C01835=1217.029,90.676,-47.866,-178.653,5.650,148.592
C01836=1217.025,90.925,-47.885,-178.651,5.651,148.591
C01837=1217.020,91.174,-47.903,-178.648,5.652,148.591
C01838=1217.015,91.423,-47.921,-178.645,5.653,148.590
C01839=1217.010,91.673,-47.939,-178.643,5.654,148.590
C01840=1217.005,91.922,-47.957,-178.641,5.654,148.589
C01841=1217.000,92.172,-47.976,-178.638,5.655,148.588
C01842=1216.996,92.421,-47.994,-178.635,5.657,148.588
C01843=1216.991,92.670,-48.012,-178.633,5.657,148.587
C01844=1216.986,92.919,-48.030,-178.630,5.658,148.587
C01845=1216.982,93.169,-48.049,-178.628,5.659,148.586
C01846=1216.976,93.418,-48.067,-178.625,5.660,148.586
C01847=1216.971,93.667,-48.086,-178.622,5.661,148.585
C01848=1216.967,93.916,-48.104,-178.620,5.662,148.585
C01849=1216.962,94.166,-48.122,-178.617,5.662,148.584
C01850=1216.957,94.415,-48.140,-178.615,5.663,148.584
C01851=1216.952,94.664,-48.159,-178.612,5.665,148.583
C01852=1216.948,94.914,-48.178,-178.609,5.665,148.582
C01853=1216.943,95.163,-48.196,-178.607,5.666,148.582
C01854=1216.938,95.412,-48.214,-178.605,5.667,148.581
C01855=1216.932,95.661,-48.233,-178.601,5.668,148.581
C01856=1216.928,95.911,-48.251,-178.599,5.669,148.580
C01857=1216.923,96.160,-48.269,-178.597,5.670,148.579
C01858=1216.919,96.409,-48.288,-178.594,5.670,148.579
C01859=1216.914,96.659,-48.307,-178.592,5.671,148.578
C01860=1216.909,96.908,-48.325,-178.589,5.673,148.578
C01861=1216.904,97.156,-48.344,-178.587,5.674,148.577
C01862=1216.898,97.406,-48.362,-178.584,5.674,148.577
C01863=1216.894,97.656,-48.381,-178.581,5.675,148.576
C01864=1216.889,97.904,-48.399,-178.579,5.677,148.576
C01865=1216.884,98.154,-48.418,-178.576,5.677,148.575
C01866=1216.880,98.403,-48.437,-178.573,5.678,148.574
C01867=1216.875,98.652,-48.455,-178.571,5.679,148.574
C01868=1216.869,98.902,-48.473,-178.568,5.680,148.573
C01869=1216.865,99.151,-48.492,-178.566,5.681,148.573
C01870=1216.860,99.400,-48.510,-178.563,5.682,148.572
C01871=1216.856,99.650,-48.530,-178.561,5.682,148.572
C01872=1216.851,99.899,-48.548,-178.558,5.684,148.571
C01873=1216.846,100.148,-48.567,-178.555,5.685,148.571
C01874=1216.841,100.398,-48.586,-178.553,5.686,148.570
C01875=1216.836,100.646,-48.604,-178.551,5.686,148.569
C01876=1216.831,100.896,-48.623,-178.548,5.688,148.569
C01877=1216.827,101.145,-48.642,-178.545,5.689,148.568
C01878=1216.822,101.394,-48.660,-178.543,5.689,148.568
C01879=1216.817,101.643,-48.679,-178.540,5.690,148.567
C01880=1216.812,101.893,-48.698,-178.537,5.692,148.567
C01881=1216.807,102.142,-48.717,-178.535,5.692,148.566
C01882=1216.803,102.392,-48.735,-178.533,5.693,148.566
C01883=1216.797,102.641,-48.755,-178.530,5.695,148.565
C01884=1216.792,102.890,-48.773,-178.527,5.695,148.564
C01885=1216.788,103.139,-48.792,-178.525,5.696,148.564
C01886=1216.783,103.388,-48.811,-178.522,5.697,148.563
C01887=1216.779,103.638,-48.829,-178.519,5.699,148.563
C01888=1216.773,103.887,-48.849,-178.517,5.699,148.562
C01889=1216.769,104.137,-48.867,-178.514,5.700,148.562
C01890=1216.764,104.385,-48.886,-178.512,5.702,148.561
C01891=1216.759,104.634,-48.905,-178.509,5.702,148.561
C01892=1216.754,104.884,-48.924,-178.507,5.703,148.560
C01893=1216.749,105.133,-48.943,-178.504,5.704,148.559
C01894=1216.745,105.382,-48.962,-178.502,5.705,148.559
C01895=1216.740,105.631,-48.980,-178.499,5.706,148.558
C01896=1216.735,105.881,-49.000,-178.496,5.707,148.558
C01897=1216.730,106.130,-49.019,-178.494,5.708,148.557
C01898=1216.725,106.380,-49.037,-178.491,5.709,148.557
C01899=1216.721,106.628,-49.056,-178.489,5.710,148.556
C01900=1216.715,106.877,-49.075,-178.486,5.711,148.556
C01901=1216.710,107.146,-49.096,-178.483,5.712,148.555
C01902=1216.705,107.414,-49.116,-178.481,5.713,148.555
C01903=1216.700,107.683,-49.137,-178.478,5.714,148.554
C01904=1216.695,107.951,-49.157,-178.475,5.715,148.553
C01905=1216.690,108.201,-49.177,-178.472,5.716,148.553
C01906=1216.685,108.449,-49.195,-178.470,5.717,148.552
C01907=1216.681,108.699,-49.215,-178.467,5.718,148.552
C01908=1216.676,108.948,-49.233,-178.465,5.720,148.551
C01909=1216.671,109.198,-49.253,-178.462,5.720,148.551
C01910=1216.666,109.447,-49.272,-178.460,5.721,148.550
C01911=1216.662,109.696,-49.291,-178.457,5.722,148.550
C01912=1216.656,109.945,-49.310,-178.454,5.723,148.549
C01913=1216.651,110.194,-49.330,-178.452,5.724,148.549
C01914=1216.647,110.443,-49.348,-178.449,5.725,148.548
C01915=1216.642,110.693,-49.368,-178.447,5.727,148.548
C01916=1216.638,110.942,-49.387,-178.444,5.727,148.547
C01917=1216.632,111.191,-49.406,-178.442,5.728,148.546
C01918=1216.628,111.441,-49.426,-178.439,5.730,148.546
C01919=1216.623,111.689,-49.444,-178.437,5.731,148.545
C01920=1216.618,111.939,-49.464,-178.434,5.731,148.545
C01921=1216.613,112.188,-49.483,-178.431,5.733,148.544
C01922=1216.609,112.438,-49.502,-178.429,5.734,148.544
C01923=1216.603,112.686,-49.521,-178.426,5.734,148.543
C01924=1216.599,112.936,-49.541,-178.423,5.736,148.543
C01925=1216.594,113.186,-49.560,-178.421,5.737,148.542
C01926=1216.589,113.434,-49.579,-178.419,5.738,148.542
C01927=1216.585,113.684,-49.599,-178.415,5.739,148.541
C01928=1216.579,113.933,-49.618,-178.413,5.740,148.541
C01929=1216.574,114.182,-49.638,-178.411,5.741,148.540
C01930=1216.570,114.431,-49.656,-178.407,5.742,148.539
C01931=1216.565,114.680,-49.676,-178.405,5.743,148.539
C01932=1216.560,114.930,-49.696,-178.403,5.744,148.538
C01933=1216.555,115.179,-49.715,-178.400,5.745,148.538
C01934=1216.551,115.428,-49.734,-178.397,5.746,148.537
C01935=1216.546,115.677,-49.753,-178.395,5.747,148.537
C01936=1216.541,115.926,-49.773,-178.392,5.748,148.536
C01937=1216.536,116.176,-49.792,-178.390,5.749,148.536
C01938=1216.532,116.425,-49.811,-178.387,5.750,148.535
C01939=1216.527,116.673,-49.832,-178.385,5.752,148.535
C01940=1216.522,116.923,-49.851,-178.382,5.752,148.534
C01941=1216.517,117.172,-49.871,-178.379,5.754,148.534
C01942=1216.512,117.421,-49.890,-178.377,5.755,148.533
C01943=1216.507,117.670,-49.909,-178.375,5.756,148.533
C01944=1216.503,117.920,-49.929,-178.372,5.757,148.532
C01945=1216.498,118.169,-49.948,-178.369,5.758,148.532
C01946=1216.493,118.418,-49.967,-178.367,5.759,148.531
C01947=1216.488,118.667,-49.988,-178.364,5.760,148.531
C01948=1216.484,118.917,-50.007,-178.362,5.761,148.530
C01949=1216.478,119.165,-50.027,-178.359,5.762,148.529
C01950=1216.474,119.415,-50.046,-178.356,5.763,148.529
C01951=1216.470,119.664,-50.065,-178.354,5.764,148.528
C01952=1216.464,119.913,-50.085,-178.351,5.766,148.528
C01953=1216.460,120.162,-50.105,-178.348,5.766,148.527
C01954=1216.455,120.412,-50.125,-178.346,5.767,148.527
C01955=1216.450,120.661,-50.144,-178.343,5.769,148.526
C01956=1216.445,120.910,-50.164,-178.341,5.770,148.526
C01957=1216.441,121.159,-50.184,-178.338,5.770,148.525
C01958=1216.436,121.409,-50.204,-178.336,5.772,148.525
C01959=1216.430,121.657,-50.223,-178.333,5.773,148.524
C01960=1216.426,121.907,-50.243,-178.330,5.775,148.524
C01961=1216.422,122.156,-50.263,-178.328,5.775,148.523
C01962=1216.417,122.405,-50.282,-178.326,5.776,148.523
C01963=1216.412,122.654,-50.301,-178.322,5.778,148.522
C01964=1216.408,122.903,-50.322,-178.320,5.779,148.522
C01965=1216.403,123.153,-50.341,-178.318,5.779,148.521
C01966=1216.397,123.401,-50.361,-178.315,5.781,148.521
C01967=1216.393,123.650,-50.381,-178.312,5.782,148.520
C01968=1216.388,123.900,-50.401,-178.310,5.783,148.520
C01969=1216.383,124.150,-50.420,-178.307,5.784,148.519
C01970=1216.378,124.398,-50.440,-178.305,5.785,148.519
C01971=1216.374,124.647,-50.460,-178.302,5.786,148.518
C01972=1216.369,124.896,-50.480,-178.300,5.787,148.518
C01973=1216.365,125.146,-50.500,-178.297,5.789,148.517
C01974=1216.360,125.395,-50.520,-178.294,5.790,148.517
C01975=1216.355,125.644,-50.540,-178.292,5.791,148.516
C01976=1216.350,125.893,-50.559,-178.289,5.792,148.516
C01977=1216.346,126.142,-50.580,-178.287,5.793,148.515
C01978=1216.341,126.392,-50.599,-178.284,5.795,148.514
C01979=1216.336,126.641,-50.620,-178.282,5.796,148.514
C01980=1216.330,126.890,-50.640,-178.279,5.797,148.513
C01981=1216.326,127.139,-50.660,-178.276,5.798,148.513
C01982=1216.321,127.388,-50.680,-178.274,5.799,148.512
C01983=1216.317,127.637,-50.700,-178.271,5.800,148.512
C01984=1216.312,127.887,-50.720,-178.269,5.801,148.511
C01985=1216.307,128.135,-50.740,-178.266,5.803,148.511
C01986=1216.302,128.385,-50.759,-178.263,5.803,148.510
C01987=1216.298,128.634,-50.780,-178.261,5.804,148.510
C01988=1216.293,128.883,-50.800,-178.258,5.806,148.509
C01989=1216.289,129.132,-50.820,-178.256,5.807,148.509
C01990=1216.283,129.382,-50.840,-178.253,5.809,148.509
C01991=1216.278,129.630,-50.860,-178.251,5.809,148.508
C01992=1216.274,129.879,-50.881,-178.248,5.811,148.508
C01993=1216.269,130.129,-50.900,-178.245,5.812,148.507
C01994=1216.264,130.378,-50.921,-178.243,5.813,148.507
C01995=1216.260,130.627,-50.940,-178.240,5.814,148.506
C01996=1216.255,130.876,-50.961,-178.238,5.815,148.505
C01997=1216.250,131.126,-50.982,-178.235,5.816,148.505
C01998=1216.245,131.374,-51.001,-178.233,5.817,148.504
C01999=1216.240,131.623,-51.021,-178.229,5.819,148.504
C02000=1216.236,131.872,-51.042,-178.227,5.820,148.503
C02001=1216.231,132.122,-51.061,-178.225,5.822,148.503
C02002=1216.226,132.371,-51.082,-178.222,5.822,148.502
C02003=1216.221,132.620,-51.103,-178.220,5.823,148.502
C02004=1216.217,132.870,-51.122,-178.217,5.825,148.501
C02005=1216.211,133.138,-51.145,-178.214,5.826,148.501
C02006=1216.206,133.407,-51.166,-178.211,5.827,148.500
C02007=1216.201,133.675,-51.188,-178.208,5.829,148.500
C02008=1216.195,133.944,-51.210,-178.206,5.829,148.499
C02009=1216.191,134.193,-51.230,-178.203,5.831,148.499
C02010=1216.187,134.442,-51.251,-178.201,5.832,148.498
C02011=1216.182,134.691,-51.271,-178.198,5.833,148.498
C02012=1216.177,134.941,-51.291,-178.196,5.834,148.497
C02013=1216.172,135.190,-51.312,-178.193,5.836,148.497
C02014=1216.168,135.439,-51.332,-178.190,5.837,148.496
C02015=1216.163,135.688,-51.353,-178.188,5.839,148.496
C02016=1216.158,135.937,-51.373,-178.185,5.839,148.495
C02017=1216.153,136.186,-51.393,-178.182,5.841,148.495
C02018=1216.148,136.436,-51.414,-178.180,5.842,148.495
C02019=1216.144,136.685,-51.434,-178.177,5.843,148.494
C02020=1216.139,136.934,-51.455,-178.175,5.844,148.494
C02021=1216.134,137.183,-51.476,-178.172,5.846,148.493
C02022=1216.130,137.432,-51.496,-178.170,5.847,148.493
C02023=1216.125,137.681,-51.516,-178.167,5.847,148.492
C02024=1216.120,137.931,-51.537,-178.164,5.849,148.492
C02025=1216.115,138.180,-51.557,-178.162,5.850,148.491
C02026=1216.111,138.428,-51.577,-178.159,5.852,148.490
C02027=1216.106,138.678,-51.598,-178.157,5.853,148.490
C02028=1216.101,138.927,-51.619,-178.154,5.854,148.489
C02029=1216.097,139.176,-51.639,-178.152,5.855,148.489
C02030=1216.092,139.425,-51.660,-178.149,5.857,148.489
C02031=1216.087,139.674,-51.680,-178.146,5.857,148.488
C02032=1216.082,139.923,-51.701,-178.144,5.859,148.488
C02033=1216.078,140.172,-51.722,-178.141,5.860,148.487
C02034=1216.073,140.421,-51.743,-178.139,5.862,148.487
C02035=1216.068,140.670,-51.763,-178.136,5.863,148.486
C02036=1216.064,140.919,-51.783,-178.133,5.864,148.486
C02037=1216.059,141.168,-51.804,-178.131,5.865,148.485
C02038=1216.054,141.417,-51.825,-178.128,5.867,148.485
C02039=1216.049,141.667,-51.846,-178.126,5.867,148.484
C02040=1216.044,141.916,-51.866,-178.123,5.869,148.484
C02041=1216.039,142.165,-51.887,-178.121,5.870,148.483
C02042=1216.035,142.414,-51.907,-178.118,5.872,148.483
C02043=1216.030,142.663,-51.928,-178.116,5.873,148.482
C02044=1216.026,142.911,-51.949,-178.113,5.874,148.482
C02045=1216.020,143.161,-51.970,-178.111,5.875,148.481
C02046=1216.016,143.410,-51.991,-178.107,5.877,148.481
C02047=1216.011,143.660,-52.012,-178.105,5.878,148.480
C02048=1216.007,143.909,-52.033,-178.103,5.879,148.480
C02049=1216.002,144.158,-52.053,-178.100,5.880,148.479
C02050=1215.997,144.407,-52.074,-178.097,5.882,148.479
C02051=1215.992,144.656,-52.095,-178.095,5.884,148.479
C02052=1215.988,144.904,-52.116,-178.092,5.884,148.478
C02053=1215.983,145.154,-52.137,-178.089,5.886,148.478
C02054=1215.978,145.403,-52.157,-178.087,5.887,148.477
C02055=1215.973,145.652,-52.178,-178.084,5.888,148.477
C02056=1215.969,145.901,-52.199,-178.082,5.889,148.476
C02057=1215.965,146.150,-52.221,-178.079,5.891,148.476
C02058=1215.959,146.399,-52.242,-178.077,5.892,148.475
C02059=1215.955,146.648,-52.262,-178.074,5.894,148.475
C02060=1215.950,146.898,-52.283,-178.071,5.894,148.474
C02061=1215.946,147.146,-52.304,-178.069,5.896,148.474
C02062=1215.940,147.395,-52.325,-178.067,5.897,148.474
C02063=1215.935,147.644,-52.346,-178.064,5.899,148.473
C02064=1215.931,147.894,-52.367,-178.061,5.900,148.473
C02065=1215.927,148.143,-52.388,-178.058,5.901,148.472
C02066=1215.921,148.392,-52.409,-178.056,5.903,148.472
C02067=1215.917,148.641,-52.430,-178.053,5.904,148.471
C02068=1215.912,148.890,-52.451,-178.050,5.905,148.471
C02069=1215.907,149.139,-52.472,-178.048,5.906,148.470
C02070=1215.903,149.388,-52.493,-178.046,5.908,148.470
C02071=1215.898,149.637,-52.515,-178.043,5.909,148.469
C02072=1215.893,149.886,-52.536,-178.040,5.910,148.469
C02073=1215.889,150.135,-52.557,-178.038,5.911,148.468
C02074=1215.884,150.384,-52.578,-178.035,5.913,148.468
C02075=1215.879,150.634,-52.599,-178.033,5.914,148.467
C02076=1215.875,150.882,-52.620,-178.030,5.916,148.467
C02077=1215.870,151.132,-52.641,-178.027,5.917,148.466
C02078=1215.865,151.380,-52.663,-178.025,5.918,148.466
C02079=1215.860,151.629,-52.684,-178.022,5.920,148.466
C02080=1215.856,151.879,-52.705,-178.020,5.921,148.465
C02081=1215.851,152.128,-52.726,-178.017,5.922,148.465
C02082=1215.846,152.377,-52.747,-178.015,5.923,148.464
C02083=1215.841,152.626,-52.769,-178.012,5.925,148.464
C02084=1215.837,152.875,-52.790,-178.009,5.927,148.463
C02085=1215.832,153.124,-52.811,-178.007,5.928,148.463
C02086=1215.827,153.373,-52.832,-178.004,5.929,148.462
C02087=1215.822,153.622,-52.854,-178.002,5.930,148.462
C02088=1215.818,153.871,-52.875,-177.999,5.932,148.462
C02089=1215.814,154.120,-52.896,-177.997,5.933,148.461
C02090=1215.809,154.369,-52.918,-177.994,5.934,148.461
C02091=1215.804,154.618,-52.939,-177.991,5.936,148.460
C02092=1215.799,154.867,-52.961,-177.989,5.937,148.460
C02093=1215.795,155.116,-52.981,-177.986,5.939,148.459
C02094=1215.790,155.365,-53.003,-177.984,5.940,148.459
C02095=1215.785,155.614,-53.024,-177.981,5.941,148.458
C02096=1215.781,155.864,-53.046,-177.978,5.943,148.458
C02097=1215.776,156.112,-53.068,-177.976,5.944,148.457
C02098=1215.770,156.361,-53.089,-177.973,5.946,148.457
C02099=1215.766,156.611,-53.111,-177.971,5.946,148.456
C02100=1215.762,156.859,-53.132,-177.968,5.948,148.456
C02101=1215.757,157.108,-53.153,-177.965,5.950,148.456
C02102=1215.753,157.358,-53.175,-177.963,5.951,148.455
C02103=1215.748,157.606,-53.197,-177.960,5.952,148.455
C02104=1215.743,157.856,-53.218,-177.958,5.953,148.454
C02105=1215.738,158.105,-53.240,-177.955,5.955,148.454
C02106=1215.733,158.354,-53.261,-177.952,5.957,148.453
C02107=1215.728,158.603,-53.282,-177.950,5.958,148.453
C02108=1215.724,158.852,-53.304,-177.947,5.959,148.453
C02109=1215.719,159.121,-53.327,-177.944,5.961,148.452
C02110=1215.714,159.390,-53.351,-177.942,5.962,148.452
C02111=1215.709,159.659,-53.374,-177.939,5.963,148.451
C02112=1215.704,159.928,-53.397,-177.936,5.965,148.451
C02113=1215.699,160.177,-53.419,-177.934,5.967,148.450
C02114=1215.694,160.426,-53.441,-177.931,5.968,148.450
C02115=1215.690,160.675,-53.463,-177.928,5.969,148.449
C02116=1215.685,160.924,-53.484,-177.926,5.971,148.449
C02117=1215.680,161.174,-53.506,-177.924,5.972,148.448
C02118=1215.676,161.422,-53.527,-177.920,5.974,148.448
C02119=1215.671,161.671,-53.549,-177.918,5.975,148.447
C02120=1215.666,161.920,-53.571,-177.916,5.976,148.447
C02121=1215.662,162.169,-53.593,-177.913,5.978,148.447
C02122=1215.657,162.418,-53.615,-177.910,5.979,148.446
C02123=1215.652,162.667,-53.637,-177.908,5.981,148.446
C02124=1215.648,162.915,-53.658,-177.905,5.982,148.445
C02125=1215.643,163.165,-53.680,-177.902,5.983,148.445
C02126=1215.638,163.414,-53.701,-177.900,5.985,148.444
C02127=1215.634,163.663,-53.723,-177.897,5.987,148.444
C02128=1215.629,163.912,-53.745,-177.895,5.988,148.444
C02129=1215.624,164.161,-53.767,-177.892,5.989,148.443
C02130=1215.620,164.410,-53.789,-177.889,5.991,148.443
C02131=1215.615,164.659,-53.810,-177.887,5.992,148.442
C02132=1215.611,164.908,-53.832,-177.884,5.994,148.442
C02133=1215.605,165.157,-53.855,-177.882,5.994,148.441
C02134=1215.601,165.406,-53.877,-177.879,5.996,148.441
C02135=1215.596,165.655,-53.898,-177.877,5.998,148.441
C02136=1215.592,165.904,-53.921,-177.874,5.999,148.440
C02137=1215.587,166.153,-53.942,-177.871,6.001,148.440
C02138=1215.583,166.402,-53.964,-177.869,6.002,148.439
C02139=1215.578,166.651,-53.986,-177.867,6.003,148.439
C02140=1215.573,166.900,-54.008,-177.864,6.005,148.439
C02141=1215.568,167.149,-54.030,-177.861,6.007,148.438
C02142=1215.563,167.399,-54.052,-177.859,6.008,148.438
C02143=1215.559,167.647,-54.074,-177.856,6.009,148.437
C02144=1215.555,167.896,-54.097,-177.853,6.011,148.437
C02145=1215.550,168.145,-54.118,-177.851,6.012,148.436
C02146=1215.546,168.394,-54.140,-177.848,6.014,148.436
C02147=1215.540,168.643,-54.163,-177.845,6.016,148.435
C02148=1215.536,168.892,-54.185,-177.843,6.017,148.435
C02149=1215.531,169.141,-54.206,-177.841,6.018,148.435
C02150=1215.527,169.390,-54.229,-177.838,6.020,148.434
C02151=1215.522,169.638,-54.251,-177.835,6.021,148.434
C02152=1215.517,169.888,-54.274,-177.833,6.023,148.433
C02153=1215.512,170.136,-54.295,-177.830,6.024,148.433
C02154=1215.508,170.386,-54.317,-177.827,6.026,148.433
C02155=1215.503,170.634,-54.339,-177.825,6.027,148.432
C02156=1215.498,170.883,-54.362,-177.822,6.029,148.432
C02157=1215.493,171.132,-54.384,-177.820,6.031,148.431
C02158=1215.489,171.381,-54.406,-177.817,6.032,148.431
C02159=1215.484,171.631,-54.429,-177.815,6.033,148.431
C02160=1215.480,171.879,-54.451,-177.812,6.035,148.430
C02161=1215.475,172.128,-54.473,-177.810,6.036,148.430
C02162=1215.470,172.377,-54.495,-177.807,6.038,148.429
C02163=1215.465,172.627,-54.517,-177.804,6.039,148.429
C02164=1215.461,172.875,-54.540,-177.802,6.040,148.428
C02165=1215.457,173.124,-54.562,-177.799,6.042,148.428
C02166=1215.452,173.374,-54.585,-177.796,6.044,148.428
C02167=1215.447,173.622,-54.607,-177.794,6.046,148.427
C02168=1215.443,173.871,-54.629,-177.792,6.047,148.427
C02169=1215.437,174.120,-54.651,-177.789,6.048,148.426
C02170=1215.433,174.369,-54.674,-177.786,6.050,148.426
C02171=1215.429,174.618,-54.696,-177.784,6.051,148.425
C02172=1215.423,174.867,-54.718,-177.781,6.053,148.425
C02173=1215.419,175.116,-54.741,-177.778,6.055,148.425
C02174=1215.414,175.366,-54.764,-177.776,6.056,148.424
C02175=1215.410,175.614,-54.786,-177.774,6.057,148.424
C02176=1215.405,175.863,-54.808,-177.770,6.059,148.423
C02177=1215.400,176.111,-54.831,-177.768,6.061,148.423
C02178=1215.396,176.361,-54.853,-177.766,6.062,148.423
C02179=1215.391,176.610,-54.876,-177.763,6.063,148.422
C02180=1215.386,176.858,-54.898,-177.760,6.065,148.422
C02181=1215.382,177.108,-54.920,-177.757,6.067,148.421
C02182=1215.377,177.357,-54.944,-177.755,6.068,148.421
C02183=1215.373,177.605,-54.965,-177.752,6.070,148.421
C02184=1215.368,177.854,-54.989,-177.750,6.071,148.420
C02185=1215.364,178.104,-55.011,-177.747,6.073,148.420
C02186=1215.358,178.352,-55.034,-177.745,6.074,148.420
C02187=1215.354,178.601,-55.056,-177.742,6.076,148.419
C02188=1215.349,178.850,-55.079,-177.739,6.078,148.419
C02189=1215.345,179.099,-55.102,-177.737,6.079,148.418
C02190=1215.340,179.348,-55.124,-177.735,6.080,148.418
C02191=1215.336,179.597,-55.147,-177.732,6.082,148.418
C02192=1215.331,179.846,-55.170,-177.729,6.084,148.417
C02193=1215.326,180.094,-55.192,-177.727,6.085,148.417
C02194=1215.321,180.343,-55.215,-177.724,6.086,148.416
C02195=1215.317,180.593,-55.237,-177.721,6.088,148.416
C02196=1215.313,180.842,-55.261,-177.719,6.090,148.415
C02197=1215.308,181.090,-55.283,-177.717,6.091,148.415
C02198=1215.303,181.339,-55.306,-177.714,6.093,148.415
C02199=1215.299,181.588,-55.329,-177.711,6.095,148.414
C02200=1215.293,181.837,-55.351,-177.708,6.096,148.414
C02201=1215.289,182.086,-55.374,-177.705,6.098,148.413
C02202=1215.285,182.335,-55.397,-177.703,6.099,148.413
C02203=1215.280,182.584,-55.420,-177.701,6.101,148.413
C02204=1215.276,182.833,-55.442,-177.698,6.103,148.412
C02205=1215.270,183.082,-55.465,-177.695,6.105,148.412
C02206=1215.266,183.330,-55.488,-177.693,6.106,148.412
C02207=1215.262,183.579,-55.512,-177.691,6.107,148.411
C02208=1215.257,183.829,-55.534,-177.688,6.109,148.411
C02209=1215.252,184.077,-55.557,-177.685,6.111,148.410
C02210=1215.248,184.326,-55.580,-177.683,6.112,148.410
C02211=1215.244,184.575,-55.603,-177.680,6.114,148.410
C02212=1215.239,184.824,-55.625,-177.677,6.115,148.409
C02213=1215.234,185.094,-55.651,-177.675,6.117,148.409
C02214=1215.229,185.363,-55.676,-177.672,6.119,148.408
C02215=1215.224,185.633,-55.701,-177.669,6.120,148.408
C02216=1215.218,185.903,-55.726,-177.666,6.122,148.408
C02217=1215.214,186.151,-55.748,-177.664,6.124,148.407
C02218=1215.209,186.401,-55.771,-177.661,6.126,148.407
C02219=1215.204,186.649,-55.794,-177.659,6.127,148.406
C02220=1215.200,186.898,-55.817,-177.656,6.128,148.406
C02221=1215.195,187.147,-55.840,-177.653,6.130,148.406
C02222=1215.191,187.396,-55.864,-177.651,6.132,148.405
C02223=1215.186,187.645,-55.887,-177.648,6.134,148.405
C02224=1215.182,187.894,-55.910,-177.646,6.135,148.405
C02225=1215.177,188.142,-55.933,-177.643,6.137,148.404
C02226=1215.172,188.391,-55.956,-177.641,6.139,148.404
C02227=1215.167,188.640,-55.979,-177.638,6.140,148.404
C02228=1215.163,188.889,-56.002,-177.635,6.142,148.403
C02229=1215.159,189.138,-56.025,-177.633,6.143,148.403
C02230=1215.154,189.387,-56.049,-177.630,6.145,148.402
C02231=1215.149,189.636,-56.072,-177.627,6.147,148.402
C02232=1215.145,189.885,-56.096,-177.625,6.148,148.402
C02233=1215.140,190.133,-56.118,-177.622,6.150,148.401
C02234=1215.135,190.382,-56.141,-177.619,6.152,148.401
C02235=1215.131,190.631,-56.165,-177.617,6.153,148.400
C02236=1215.126,190.880,-56.188,-177.615,6.155,148.400
C02237=1215.121,191.129,-56.211,-177.612,6.157,148.400
C02238=1215.117,191.378,-56.234,-177.609,6.159,148.399
C02239=1215.113,191.627,-56.258,-177.607,6.160,148.399
C02240=1215.108,191.876,-56.281,-177.604,6.161,148.398
C02241=1215.103,192.125,-56.304,-177.601,6.163,148.398
C02242=1215.098,192.374,-56.328,-177.599,6.165,148.398
C02243=1215.094,192.622,-56.352,-177.596,6.167,148.397
C02244=1215.089,192.871,-56.375,-177.594,6.168,148.397
C02245=1215.084,193.120,-56.398,-177.591,6.170,148.397
C02246=1215.080,193.369,-56.421,-177.589,6.171,148.396
C02247=1215.075,193.618,-56.444,-177.586,6.173,148.396
C02248=1215.071,193.867,-56.467,-177.583,6.175,148.396
C02249=1215.066,194.115,-56.492,-177.581,6.177,148.395
C02250=1215.062,194.364,-56.515,-177.578,6.179,148.395
C02251=1215.057,194.613,-56.538,-177.576,6.180,148.395
C02252=1215.052,194.862,-56.562,-177.573,6.181,148.394
C02253=1215.048,195.110,-56.586,-177.571,6.183,148.394
C02254=1215.043,195.360,-56.609,-177.568,6.185,148.394
C02255=1215.038,195.609,-56.632,-177.565,6.187,148.393
C02256=1215.034,195.858,-56.656,-177.562,6.188,148.393
C02257=1215.029,196.106,-56.680,-177.560,6.190,148.392
C02258=1215.025,196.355,-56.703,-177.557,6.192,148.392
C02259=1215.020,196.604,-56.727,-177.555,6.193,148.392
C02260=1215.015,196.852,-56.751,-177.552,6.195,148.391
C02261=1215.011,197.102,-56.774,-177.550,6.197,148.391
C02262=1215.006,197.351,-56.797,-177.547,6.199,148.391
C02263=1215.002,197.599,-56.821,-177.544,6.200,148.390
C02264=1214.997,197.848,-56.845,-177.542,6.202,148.390
C02265=1214.992,198.097,-56.868,-177.539,6.204,148.389
C02266=1214.988,198.345,-56.892,-177.537,6.205,148.389
C02267=1214.983,198.594,-56.916,-177.534,6.207,148.389
C02268=1214.979,198.844,-56.939,-177.532,6.209,148.388
C02269=1214.974,199.092,-56.963,-177.529,6.211,148.388
C02270=1214.970,199.342,-56.987,-177.526,6.212,148.388
C02271=1214.966,199.590,-57.011,-177.524,6.214,148.387
C02272=1214.961,199.839,-57.034,-177.521,6.216,148.387
C02273=1214.957,200.088,-57.058,-177.519,6.218,148.387
C02274=1214.952,200.337,-57.082,-177.516,6.219,148.386
C02275=1214.947,200.585,-57.106,-177.514,6.221,148.386
C02276=1214.942,200.834,-57.130,-177.511,6.223,148.386
C02277=1214.937,201.083,-57.153,-177.509,6.224,148.385
C02278=1214.933,201.332,-57.177,-177.506,6.226,148.385
C02279=1214.929,201.580,-57.201,-177.503,6.228,148.385
C02280=1214.924,201.829,-57.225,-177.501,6.230,148.384
C02281=1214.919,202.078,-57.249,-177.498,6.232,148.384
C02282=1214.915,202.327,-57.272,-177.495,6.234,148.384
C02283=1214.911,202.576,-57.296,-177.493,6.235,148.383
C02284=1214.905,202.825,-57.320,-177.491,6.236,148.383
C02285=1214.901,203.074,-57.344,-177.488,6.238,148.383
C02286=1214.896,203.323,-57.368,-177.485,6.240,148.382
C02287=1214.892,203.571,-57.392,-177.483,6.242,148.382
C02288=1214.888,203.819,-57.416,-177.480,6.244,148.382
C02289=1214.882,204.069,-57.440,-177.477,6.246,148.381
C02290=1214.878,204.318,-57.464,-177.475,6.247,148.381
C02291=1214.874,204.566,-57.488,-177.472,6.249,148.380
C02292=1214.869,204.815,-57.512,-177.469,6.251,148.380
C02293=1214.865,205.064,-57.536,-177.467,6.253,148.380
C02294=1214.860,205.312,-57.561,-177.465,6.254,148.379
C02295=1214.855,205.561,-57.584,-177.462,6.256,148.379
C02296=1214.851,205.811,-57.608,-177.459,6.258,148.379
C02297=1214.847,206.059,-57.632,-177.457,6.260,148.378
C02298=1214.841,206.308,-57.656,-177.454,6.261,148.378
C02299=1214.837,206.557,-57.680,-177.451,6.263,148.378
C02300=1214.833,206.805,-57.704,-177.449,6.265,148.377
C02301=1214.828,207.055,-57.730,-177.446,6.267,148.377
C02302=1214.823,207.304,-57.753,-177.444,6.269,148.377
C02303=1214.819,207.552,-57.777,-177.441,6.271,148.376
C02304=1214.815,207.800,-57.801,-177.438,6.272,148.376
C02305=1214.809,208.049,-57.826,-177.436,6.274,148.376
C02306=1214.806,208.298,-57.850,-177.433,6.276,148.375
C02307=1214.801,208.547,-57.873,-177.430,6.278,148.375
C02308=1214.796,208.796,-57.898,-177.428,6.279,148.375
C02309=1214.791,209.044,-57.922,-177.426,6.281,148.374
C02310=1214.786,209.293,-57.947,-177.423,6.283,148.374
C02311=1214.783,209.542,-57.971,-177.420,6.284,148.374
C02312=1214.778,209.791,-57.995,-177.418,6.286,148.373
C02313=1214.773,210.039,-58.020,-177.415,6.288,148.373
C02314=1214.768,210.288,-58.043,-177.412,6.290,148.373
C02315=1214.765,210.538,-58.068,-177.410,6.292,148.372
C02316=1214.759,210.786,-58.093,-177.407,6.294,148.372
C02317=1214.754,211.056,-58.119,-177.405,6.296,148.372
C02318=1214.750,211.326,-58.145,-177.402,6.297,148.371
C02319=1214.745,211.597,-58.172,-177.399,6.300,148.371
C02320=1214.740,211.868,-58.198,-177.396,6.302,148.371
C02321=1214.735,212.116,-58.223,-177.393,6.304,148.370
C02322=1214.730,212.365,-58.247,-177.391,6.306,148.370
C02323=1214.727,212.614,-58.272,-177.388,6.307,148.370
C02324=1214.721,212.863,-58.296,-177.386,6.309,148.369
C02325=1214.717,213.111,-58.320,-177.383,6.311,148.369
C02326=1214.712,213.361,-58.345,-177.380,6.313,148.369
C02327=1214.708,213.609,-58.370,-177.378,6.315,148.368
C02328=1214.703,213.858,-58.394,-177.375,6.317,148.368
C02329=1214.699,214.106,-58.419,-177.372,6.318,148.368
C02330=1214.694,214.355,-58.444,-177.370,6.320,148.367
C02331=1214.690,214.604,-58.468,-177.367,6.322,148.367
C02332=1214.685,214.853,-58.493,-177.365,6.324,148.367
C02333=1214.681,215.101,-58.517,-177.362,6.326,148.367
C02334=1214.676,215.350,-58.542,-177.360,6.328,148.366
C02335=1214.672,215.599,-58.566,-177.358,6.329,148.366
C02336=1214.667,215.848,-58.591,-177.355,6.331,148.366
C02337=1214.663,216.096,-58.615,-177.352,6.333,148.365
C02338=1214.658,216.345,-58.641,-177.350,6.335,148.365
C02339=1214.653,216.594,-58.665,-177.347,6.336,148.365
C02340=1214.649,216.842,-58.690,-177.344,6.338,148.364
C02341=1214.644,217.092,-58.715,-177.342,6.340,148.364
C02342=1214.640,217.340,-58.739,-177.339,6.342,148.364
C02343=1214.636,217.589,-58.764,-177.336,6.344,148.363
C02344=1214.630,217.838,-58.789,-177.334,6.346,148.363
C02345=1214.626,218.086,-58.813,-177.332,6.348,148.363
C02346=1214.622,218.335,-58.838,-177.329,6.350,148.362
C02347=1214.617,218.583,-58.863,-177.326,6.352,148.362
C02348=1214.613,218.833,-58.888,-177.324,6.353,148.362
C02349=1214.608,219.081,-58.913,-177.321,6.355,148.361
C02350=1214.603,219.330,-58.937,-177.318,6.357,148.361
C02351=1214.599,219.579,-58.962,-177.316,6.359,148.361
C02352=1214.594,219.827,-58.987,-177.313,6.361,148.360
C02353=1214.590,220.076,-59.012,-177.311,6.363,148.360
C02354=1214.585,220.325,-59.037,-177.308,6.365,148.360
C02355=1214.581,220.574,-59.062,-177.306,6.367,148.360
C02356=1214.577,220.822,-59.087,-177.303,6.368,148.359
C02357=1214.572,221.071,-59.112,-177.301,6.370,148.359
C02358=1214.567,221.320,-59.137,-177.298,6.372,148.359
C02359=1214.563,221.568,-59.161,-177.295,6.374,148.358
C02360=1214.559,221.817,-59.186,-177.293,6.376,148.358
C02361=1214.554,222.065,-59.212,-177.290,6.378,148.358
C02362=1214.549,222.315,-59.237,-177.288,6.380,148.358
C02363=1214.545,222.563,-59.261,-177.285,6.383,148.357
C02364=1214.541,222.812,-59.287,-177.282,6.384,148.357
C02365=1214.535,223.061,-59.311,-177.279,6.386,148.357
C02366=1214.531,223.309,-59.337,-177.277,6.388,148.356
C02367=1214.527,223.558,-59.361,-177.274,6.390,148.356
C02368=1214.523,223.807,-59.387,-177.271,6.392,148.356
C02369=1214.517,224.055,-59.412,-177.269,6.394,148.356
C02370=1214.513,224.304,-59.437,-177.267,6.396,148.355
C02371=1214.508,224.553,-59.462,-177.264,6.398,148.355
C02372=1214.505,224.801,-59.487,-177.261,6.400,148.355
C02373=1214.499,225.050,-59.512,-177.259,6.401,148.354
C02374=1214.495,225.299,-59.537,-177.256,6.403,148.354
C02375=1214.490,225.547,-59.563,-177.254,6.405,148.354
C02376=1214.486,225.796,-59.588,-177.251,6.407,148.354
C02377=1214.481,226.045,-59.613,-177.249,6.409,148.353
C02378=1214.477,226.294,-59.638,-177.246,6.411,148.353
C02379=1214.473,226.542,-59.663,-177.244,6.413,148.353
C02380=1214.468,226.791,-59.689,-177.241,6.415,148.352
C02381=1214.464,227.040,-59.714,-177.238,6.417,148.352
C02382=1214.459,227.288,-59.739,-177.236,6.419,148.352
C02383=1214.455,227.537,-59.765,-177.233,6.421,148.351
C02384=1214.450,227.786,-59.790,-177.231,6.422,148.351
C02385=1214.445,228.034,-59.815,-177.228,6.424,148.351
C02386=1214.441,228.283,-59.841,-177.226,6.426,148.351
C02387=1214.437,228.532,-59.865,-177.223,6.428,148.350
C02388=1214.432,228.780,-59.891,-177.221,6.430,148.350
C02389=1214.428,229.029,-59.916,-177.218,6.432,148.350
C02390=1214.423,229.278,-59.941,-177.216,6.434,148.349
C02391=1214.419,229.527,-59.967,-177.213,6.436,148.349
C02392=1214.414,229.775,-59.993,-177.211,6.438,148.349
C02393=1214.410,230.024,-60.018,-177.208,6.440,148.349
C02394=1214.405,230.272,-60.044,-177.205,6.442,148.348
C02395=1214.400,230.521,-60.069,-177.202,6.444,148.348
C02396=1214.396,230.770,-60.095,-177.200,6.446,148.348
C02397=1214.391,231.018,-60.120,-177.198,6.448,148.348
C02398=1214.387,231.267,-60.146,-177.195,6.450,148.347
C02399=1214.383,231.516,-60.171,-177.192,6.452,148.347
C02400=1214.378,231.764,-60.196,-177.190,6.454,148.347
C02401=1214.374,232.013,-60.222,-177.187,6.456,148.346
C02402=1214.369,232.261,-60.247,-177.185,6.458,148.346
C02403=1214.365,232.510,-60.273,-177.182,6.460,148.346
C02404=1214.360,232.759,-60.299,-177.180,6.462,148.346
C02405=1214.356,233.007,-60.324,-177.177,6.463,148.345
C02406=1214.351,233.256,-60.350,-177.174,6.465,148.345
C02407=1214.347,233.505,-60.376,-177.172,6.467,148.345
C02408=1214.342,233.753,-60.402,-177.170,6.469,148.345
C02409=1214.337,234.002,-60.427,-177.167,6.471,148.344
C02410=1214.333,234.251,-60.453,-177.164,6.473,148.344
C02411=1214.329,234.500,-60.479,-177.162,6.476,148.344
C02412=1214.324,234.748,-60.504,-177.159,6.478,148.344
C02413=1214.320,234.996,-60.530,-177.156,6.480,148.343
C02414=1214.316,235.245,-60.556,-177.154,6.482,148.343
C02415=1214.311,235.493,-60.581,-177.152,6.484,148.343
C02416=1214.307,235.742,-60.607,-177.149,6.486,148.342
C02417=1214.302,235.991,-60.633,-177.146,6.488,148.342
C02418=1214.297,236.240,-60.659,-177.144,6.489,148.342
C02419=1214.292,236.488,-60.684,-177.142,6.492,148.342
C02420=1214.288,236.737,-60.710,-177.139,6.493,148.341
C02421=1214.284,237.009,-60.738,-177.136,6.496,148.341
C02422=1214.279,237.279,-60.767,-177.133,6.498,148.341
C02423=1214.274,237.551,-60.795,-177.131,6.500,148.341
C02424=1214.269,237.823,-60.822,-177.127,6.503,148.340
C02425=1214.264,238.072,-60.849,-177.125,6.504,148.340
C02426=1214.260,238.320,-60.875,-177.123,6.507,148.340
C02427=1214.255,238.569,-60.901,-177.120,6.508,148.339
C02428=1214.251,238.817,-60.927,-177.117,6.510,148.339
C02429=1214.246,239.066,-60.953,-177.115,6.512,148.339
C02430=1214.241,239.315,-60.978,-177.113,6.514,148.339
C02431=1214.237,239.563,-61.004,-177.110,6.516,148.338
C02432=1214.233,239.812,-61.030,-177.107,6.519,148.338
C02433=1214.228,240.060,-61.056,-177.105,6.521,148.338
C02434=1214.224,240.309,-61.082,-177.102,6.523,148.338
C02435=1214.219,240.558,-61.108,-177.099,6.525,148.337
C02436=1214.215,240.806,-61.134,-177.097,6.527,148.337
C02437=1214.210,241.055,-61.161,-177.095,6.529,148.337
C02438=1214.206,241.304,-61.187,-177.092,6.531,148.337
C02439=1214.202,241.551,-61.213,-177.089,6.533,148.336
C02440=1214.197,241.800,-61.239,-177.087,6.535,148.336
C02441=1214.193,242.049,-61.265,-177.084,6.537,148.336
C02442=1214.188,242.298,-61.290,-177.081,6.539,148.336
C02443=1214.184,242.547,-61.318,-177.079,6.541,148.336
C02444=1214.179,242.795,-61.343,-177.077,6.543,148.335
C02445=1214.175,243.043,-61.369,-177.074,6.545,148.335
C02446=1214.170,243.292,-61.396,-177.071,6.547,148.335
C02447=1214.166,243.541,-61.422,-177.069,6.549,148.335
C02448=1214.161,243.789,-61.449,-177.067,6.551,148.334
C02449=1214.157,244.038,-61.474,-177.063,6.554,148.334
C02450=1214.153,244.287,-61.500,-177.061,6.556,148.334
C02451=1214.148,244.535,-61.527,-177.059,6.558,148.334
C02452=1214.143,244.783,-61.553,-177.056,6.560,148.333
C02453=1214.138,245.032,-61.580,-177.054,6.562,148.333
C02454=1214.134,245.281,-61.605,-177.051,6.564,148.333
C02455=1214.130,245.529,-61.632,-177.049,6.566,148.333
C02456=1214.125,245.778,-61.658,-177.046,6.569,148.333
C02457=1214.121,246.026,-61.685,-177.043,6.570,148.332
C02458=1214.116,246.275,-61.711,-177.041,6.572,148.332
C02459=1214.113,246.523,-61.737,-177.039,6.575,148.332
C02460=1214.108,246.773,-61.764,-177.036,6.576,148.331
C02461=1214.104,247.021,-61.790,-177.033,6.578,148.331
C02462=1214.099,247.270,-61.817,-177.031,6.580,148.331
C02463=1214.095,247.518,-61.843,-177.028,6.583,148.331
C02464=1214.090,247.766,-61.870,-177.025,6.585,148.330
C02465=1214.085,248.015,-61.895,-177.023,6.587,148.330
C02466=1214.081,248.263,-61.923,-177.021,6.589,148.330
C02467=1214.076,248.512,-61.948,-177.018,6.591,148.330
C02468=1214.072,248.760,-61.975,-177.016,6.593,148.330
C02469=1214.068,249.009,-62.002,-177.013,6.595,148.329
C02470=1214.063,249.258,-62.028,-177.010,6.598,148.329
C02471=1214.059,249.506,-62.055,-177.008,6.600,148.329
C02472=1214.054,249.754,-62.082,-177.005,6.602,148.329
C02473=1214.050,250.003,-62.107,-177.003,6.604,148.329
C02474=1214.045,250.252,-62.135,-177.001,6.606,148.328
C02475=1214.041,250.500,-62.162,-176.998,6.608,148.328
C02476=1214.037,250.749,-62.187,-176.995,6.611,148.328
C02477=1214.032,250.998,-62.214,-176.993,6.613,148.328
C02478=1214.028,251.246,-62.241,-176.990,6.614,148.327
C02479=1214.023,251.494,-62.268,-176.988,6.617,148.327
C02480=1214.018,251.743,-62.294,-176.985,6.618,148.327
C02481=1214.014,251.992,-62.321,-176.983,6.621,148.327
C02482=1214.010,252.240,-62.348,-176.980,6.623,148.327
C02483=1214.006,252.488,-62.374,-176.977,6.625,148.326
C02484=1214.001,252.737,-62.401,-176.975,6.627,148.326
C02485=1213.996,252.986,-62.428,-176.973,6.629,148.326
C02486=1213.992,253.234,-62.454,-176.970,6.631,148.326
C02487=1213.988,253.483,-62.481,-176.967,6.634,148.326
C02488=1213.983,253.731,-62.508,-176.965,6.636,148.325
C02489=1213.979,253.979,-62.535,-176.963,6.638,148.325
C02490=1213.974,254.228,-62.561,-176.960,6.640,148.325
C02491=1213.970,254.478,-62.588,-176.957,6.642,148.324
C02492=1213.965,254.726,-62.616,-176.955,6.645,148.324
C02493=1213.961,254.974,-62.642,-176.952,6.647,148.324
C02494=1213.957,255.223,-62.669,-176.950,6.649,148.324
C02495=1213.952,255.471,-62.696,-176.947,6.651,148.324
C02496=1213.948,255.719,-62.723,-176.945,6.653,148.324
C02497=1213.944,255.968,-62.750,-176.942,6.656,148.323
C02498=1213.939,256.216,-62.777,-176.939,6.658,148.323
C02499=1213.934,256.465,-62.804,-176.937,6.660,148.323
C02500=1213.930,256.713,-62.830,-176.935,6.662,148.323
C02501=1213.926,256.962,-62.857,-176.932,6.665,148.323
C02502=1213.922,257.211,-62.885,-176.929,6.667,148.322
C02503=1213.917,257.459,-62.912,-176.927,6.668,148.322
C02504=1213.912,257.708,-62.939,-176.924,6.671,148.322
C02505=1213.908,257.956,-62.965,-176.922,6.672,148.322
C02506=1213.904,258.204,-62.992,-176.919,6.675,148.322
C02507=1213.899,258.453,-63.019,-176.917,6.677,148.321
C02508=1213.894,258.701,-63.047,-176.914,6.680,148.321
C02509=1213.890,258.950,-63.074,-176.912,6.681,148.321
C02510=1213.886,259.199,-63.101,-176.909,6.684,148.321
C02511=1213.882,259.447,-63.127,-176.906,6.686,148.321
C02512=1213.877,259.695,-63.155,-176.904,6.688,148.320
C02513=1213.873,259.944,-63.182,-176.902,6.690,148.320
C02514=1213.868,260.192,-63.209,-176.899,6.692,148.320
C02515=1213.864,260.441,-63.236,-176.896,6.695,148.320
C02516=1213.859,260.690,-63.264,-176.894,6.697,148.320
C02517=1213.855,260.938,-63.291,-176.892,6.699,148.319
C02518=1213.850,261.186,-63.319,-176.889,6.701,148.319
C02519=1213.846,261.435,-63.346,-176.886,6.704,148.319
C02520=1213.842,261.683,-63.372,-176.884,6.706,148.319
C02521=1213.838,261.932,-63.400,-176.882,6.708,148.319
C02522=1213.833,262.181,-63.427,-176.879,6.710,148.318
C02523=1213.829,262.428,-63.454,-176.876,6.713,148.318
C02524=1213.824,262.677,-63.482,-176.874,6.715,148.318
C02525=1213.819,262.950,-63.512,-176.871,6.717,148.318
C02526=1213.815,263.223,-63.542,-176.868,6.720,148.318
C02527=1213.810,263.495,-63.572,-176.865,6.723,148.317
C02528=1213.805,263.768,-63.601,-176.863,6.725,148.317
C02529=1213.801,264.016,-63.629,-176.860,6.727,148.317
C02530=1213.796,264.265,-63.656,-176.857,6.729,148.317
C02531=1213.792,264.514,-63.684,-176.855,6.732,148.317
C02532=1213.787,264.762,-63.711,-176.853,6.733,148.316
C02533=1213.783,265.010,-63.738,-176.850,6.737,148.316
C02534=1213.778,265.258,-63.766,-176.847,6.738,148.316
C02535=1213.774,265.507,-63.794,-176.845,6.741,148.316
C02536=1213.770,265.756,-63.821,-176.843,6.742,148.316
C02537=1213.765,266.004,-63.849,-176.840,6.745,148.316
C02538=1213.761,266.253,-63.876,-176.837,6.747,148.315
C02539=1213.756,266.501,-63.904,-176.835,6.750,148.315
C02540=1213.752,266.749,-63.931,-176.832,6.751,148.315
C02541=1213.747,266.997,-63.959,-176.830,6.754,148.315
C02542=1213.743,267.246,-63.986,-176.827,6.756,148.315
C02543=1213.739,267.494,-64.014,-176.825,6.758,148.315
C02544=1213.734,267.743,-64.041,-176.822,6.762,148.315
C02545=1213.730,267.991,-64.069,-176.820,6.763,148.314
C02546=1213.726,268.240,-64.097,-176.818,6.766,148.314
C02547=1213.721,268.488,-64.125,-176.815,6.767,148.314
C02548=1213.717,268.737,-64.152,-176.812,6.770,148.314
C02549=1213.712,268.985,-64.180,-176.810,6.772,148.314
C02550=1213.708,269.234,-64.207,-176.808,6.775,148.313
C02551=1213.704,269.482,-64.235,-176.804,6.777,148.313
C02552=1213.699,269.731,-64.262,-176.802,6.779,148.313
C02553=1213.695,269.979,-64.290,-176.800,6.781,148.313
C02554=1213.690,270.228,-64.319,-176.798,6.784,148.313
C02555=1213.686,270.476,-64.346,-176.795,6.787,148.313
C02556=1213.681,270.724,-64.374,-176.792,6.788,148.312
C02557=1213.678,270.972,-64.402,-176.790,6.791,148.312
C02558=1213.673,271.221,-64.429,-176.787,6.793,148.312
C02559=1213.668,271.469,-64.457,-176.785,6.796,148.312
C02560=1213.664,271.718,-64.485,-176.782,6.797,148.312
C02561=1213.659,271.966,-64.512,-176.780,6.800,148.312
C02562=1213.656,272.215,-64.541,-176.777,6.802,148.311
C02563=1213.651,272.463,-64.569,-176.775,6.805,148.311
C02564=1213.646,272.711,-64.596,-176.772,6.808,148.311
C02565=1213.642,272.960,-64.624,-176.769,6.809,148.311
C02566=1213.638,273.208,-64.652,-176.767,6.812,148.311
C02567=1213.633,273.457,-64.681,-176.764,6.814,148.311
C02568=1213.629,273.705,-64.709,-176.762,6.817,148.311
C02569=1213.625,273.954,-64.736,-176.760,6.819,148.311
C02570=1213.620,274.202,-64.764,-176.757,6.821,148.310
C02571=1213.616,274.450,-64.792,-176.755,6.824,148.310
C02572=1213.612,274.699,-64.820,-176.752,6.825,148.310
C02573=1213.607,274.947,-64.849,-176.749,6.829,148.310
C02574=1213.603,275.196,-64.876,-176.747,6.831,148.310
C02575=1213.598,275.444,-64.904,-176.745,6.833,148.310
C02576=1213.594,275.693,-64.933,-176.742,6.836,148.309
C02577=1213.589,275.941,-64.960,-176.739,6.837,148.309
C02578=1213.586,276.189,-64.988,-176.737,6.840,148.309
C02579=1213.581,276.437,-65.017,-176.735,6.843,148.309
C02580=1213.577,276.686,-65.045,-176.732,6.845,148.309
C02581=1213.572,276.934,-65.073,-176.730,6.847,148.309
C02582=1213.567,277.182,-65.101,-176.727,6.850,148.309
C02583=1213.564,277.431,-65.129,-176.724,6.852,148.308
C02584=1213.559,277.679,-65.158,-176.722,6.854,148.308
C02585=1213.555,277.927,-65.186,-176.719,6.857,148.308
C02586=1213.550,278.175,-65.214,-176.717,6.859,148.308
C02587=1213.546,278.424,-65.242,-176.715,6.861,148.308
C02588=1213.542,278.673,-65.270,-176.712,6.864,148.308
C02589=1213.537,278.921,-65.299,-176.710,6.866,148.308
C02590=1213.533,279.169,-65.327,-176.708,6.868,148.308
C02591=1213.528,279.418,-65.355,-176.704,6.871,148.307
C02592=1213.525,279.666,-65.383,-176.702,6.873,148.307
C02593=1213.519,279.914,-65.412,-176.700,6.876,148.307
C02594=1213.516,280.163,-65.440,-176.697,6.878,148.307
C02595=1213.511,280.411,-65.468,-176.695,6.880,148.307
C02596=1213.507,280.660,-65.496,-176.692,6.883,148.307
C02597=1213.502,280.908,-65.525,-176.690,6.885,148.307
C02598=1213.498,281.156,-65.553,-176.687,6.887,148.306
C02599=1213.494,281.405,-65.582,-176.685,6.890,148.306
C02600=1213.490,281.653,-65.610,-176.682,6.892,148.306
C02601=1213.485,281.901,-65.639,-176.680,6.894,148.306
C02602=1213.481,282.149,-65.667,-176.677,6.897,148.306
C02603=1213.476,282.398,-65.695,-176.675,6.899,148.306
C02604=1213.472,282.645,-65.724,-176.672,6.902,148.306
C02605=1213.468,282.894,-65.753,-176.670,6.904,148.306
C02606=1213.463,283.143,-65.781,-176.667,6.906,148.305
C02607=1213.459,283.391,-65.809,-176.665,6.909,148.305
C02608=1213.454,283.640,-65.838,-176.662,6.912,148.305
C02609=1213.450,283.887,-65.866,-176.660,6.915,148.305
C02610=1213.446,284.136,-65.895,-176.657,6.916,148.305
C02611=1213.441,284.385,-65.924,-176.655,6.919,148.305
C02612=1213.437,284.632,-65.952,-176.652,6.922,148.305
C02613=1213.433,284.881,-65.981,-176.650,6.924,148.305
C02614=1213.428,285.129,-66.010,-176.647,6.927,148.305
C02615=1213.424,285.377,-66.038,-176.645,6.929,148.304
C02616=1213.420,285.626,-66.067,-176.643,6.931,148.304
C02617=1213.415,285.874,-66.096,-176.640,6.934,148.304
C02618=1213.411,286.122,-66.124,-176.638,6.936,148.304
C02619=1213.407,286.371,-66.153,-176.635,6.939,148.304
C02620=1213.402,286.619,-66.181,-176.633,6.941,148.304
C02621=1213.398,286.867,-66.210,-176.630,6.943,148.304
C02622=1213.394,287.116,-66.239,-176.627,6.946,148.304
C02623=1213.389,287.364,-66.268,-176.625,6.948,148.304
C02624=1213.385,287.612,-66.296,-176.623,6.951,148.304
C02625=1213.381,287.861,-66.326,-176.620,6.953,148.303
C02626=1213.376,288.109,-66.354,-176.618,6.955,148.303
C02627=1213.372,288.357,-66.384,-176.615,6.958,148.303
C02628=1213.368,288.606,-66.412,-176.613,6.961,148.303
C02629=1213.362,288.880,-66.444,-176.610,6.963,148.303
C02630=1213.358,289.154,-66.476,-176.607,6.966,148.303
C02631=1213.353,289.428,-66.508,-176.604,6.969,148.303
C02632=1213.348,289.703,-66.540,-176.602,6.971,148.303
C02633=1213.344,289.951,-66.569,-176.599,6.974,148.303
C02634=1213.340,290.199,-66.597,-176.597,6.977,148.303
C02635=1213.336,290.447,-66.626,-176.595,6.980,148.303
C02636=1213.331,290.696,-66.655,-176.592,6.981,148.302
C02637=1213.327,290.944,-66.684,-176.590,6.984,148.302
C02638=1213.322,291.192,-66.714,-176.587,6.987,148.302
C02639=1213.318,291.441,-66.742,-176.585,6.989,148.302
C02640=1213.314,291.689,-66.771,-176.582,6.992,148.302
C02641=1213.310,291.937,-66.801,-176.580,6.994,148.302
C02642=1213.305,292.185,-66.829,-176.577,6.997,148.302
C02643=1213.301,292.434,-66.858,-176.575,6.999,148.302
C02644=1213.297,292.682,-66.888,-176.573,7.001,148.302
C02645=1213.292,292.931,-66.917,-176.570,7.004,148.302
C02646=1213.287,293.178,-66.946,-176.568,7.006,148.301
C02647=1213.283,293.427,-66.975,-176.565,7.009,148.301
C02648=1213.279,293.675,-67.003,-176.563,7.011,148.301
C02649=1213.275,293.923,-67.033,-176.560,7.014,148.301
C02650=1213.271,294.172,-67.062,-176.558,7.017,148.301
C02651=1213.266,294.419,-67.091,-176.555,7.020,148.301
C02652=1213.262,294.668,-67.120,-176.553,7.022,148.301
C02653=1213.258,294.916,-67.149,-176.550,7.024,148.301
C02654=1213.253,295.165,-67.179,-176.548,7.027,148.301
C02655=1213.249,295.413,-67.208,-176.546,7.029,148.301
C02656=1213.245,295.661,-67.238,-176.543,7.032,148.301
C02657=1213.240,295.909,-67.267,-176.541,7.034,148.301
C02658=1213.236,296.158,-67.296,-176.538,7.037,148.301
C02659=1213.232,296.406,-67.325,-176.536,7.039,148.301
C02660=1213.227,296.654,-67.355,-176.533,7.042,148.300
C02661=1213.223,296.902,-67.384,-176.531,7.044,148.300
C02662=1213.219,297.151,-67.413,-176.528,7.047,148.300
C02663=1213.215,297.399,-67.443,-176.526,7.050,148.300
C02664=1213.210,297.647,-67.472,-176.524,7.052,148.300
C02665=1213.206,297.895,-67.501,-176.521,7.055,148.300
C02666=1213.202,298.143,-67.531,-176.519,7.057,148.300
C02667=1213.198,298.391,-67.560,-176.516,7.060,148.300
C02668=1213.193,298.640,-67.590,-176.514,7.062,148.300
C02669=1213.189,298.888,-67.619,-176.511,7.065,148.300
C02670=1213.185,299.136,-67.649,-176.509,7.067,148.300
C02671=1213.181,299.384,-67.678,-176.506,7.070,148.300
C02672=1213.177,299.633,-67.708,-176.504,7.072,148.300
C02673=1213.171,299.881,-67.737,-176.502,7.076,148.300
C02674=1213.167,300.129,-67.767,-176.499,7.078,148.300
C02675=1213.163,300.377,-67.796,-176.497,7.081,148.300
C02676=1213.159,300.625,-67.826,-176.495,7.083,148.299
C02677=1213.154,300.874,-67.855,-176.492,7.086,148.299
C02678=1213.150,301.122,-67.885,-176.490,7.088,148.299
C02679=1213.146,301.370,-67.914,-176.488,7.090,148.299
C02680=1213.141,301.619,-67.944,-176.485,7.093,148.299
C02681=1213.137,301.867,-67.974,-176.483,7.096,148.299
C02682=1213.133,302.115,-68.003,-176.480,7.099,148.299
C02683=1213.129,302.363,-68.033,-176.478,7.101,148.299
C02684=1213.125,302.611,-68.063,-176.475,7.104,148.299
C02685=1213.120,302.859,-68.092,-176.473,7.106,148.299
C02686=1213.116,303.108,-68.122,-176.471,7.109,148.299
C02687=1213.111,303.356,-68.152,-176.469,7.111,148.299
C02688=1213.108,303.604,-68.182,-176.466,7.114,148.299
C02689=1213.103,303.852,-68.211,-176.464,7.117,148.299
C02690=1213.098,304.101,-68.241,-176.461,7.120,148.299
C02691=1213.094,304.349,-68.271,-176.459,7.122,148.299
C02692=1213.090,304.597,-68.301,-176.456,7.125,148.299
C02693=1213.086,304.845,-68.330,-176.454,7.127,148.299
C02694=1213.081,305.094,-68.360,-176.451,7.130,148.299
C02695=1213.077,305.342,-68.390,-176.449,7.132,148.299
C02696=1213.073,305.589,-68.420,-176.447,7.135,148.299
C02697=1213.069,305.838,-68.449,-176.445,7.138,148.299
C02698=1213.064,306.086,-68.480,-176.442,7.141,148.299
C02699=1213.060,306.334,-68.510,-176.440,7.143,148.299
C02700=1213.056,306.582,-68.539,-176.437,7.146,148.299
C02701=1213.051,306.831,-68.569,-176.435,7.148,148.299
C02702=1213.047,307.078,-68.599,-176.432,7.151,148.299
C02703=1213.043,307.327,-68.629,-176.430,7.153,148.299
C02704=1213.038,307.575,-68.660,-176.427,7.156,148.299
C02705=1213.034,307.823,-68.689,-176.425,7.159,148.298
C02706=1213.030,308.071,-68.718,-176.423,7.162,148.298
C02707=1213.025,308.319,-68.749,-176.421,7.164,148.298
C02708=1213.021,308.567,-68.779,-176.418,7.167,148.298
C02709=1213.017,308.815,-68.809,-176.416,7.169,148.298
C02710=1213.013,309.064,-68.839,-176.413,7.172,148.298
C02711=1213.009,309.311,-68.869,-176.411,7.174,148.298
C02712=1213.004,309.560,-68.899,-176.408,7.177,148.298
C02713=1213.000,309.808,-68.930,-176.407,7.180,148.298
C02714=1212.996,310.057,-68.960,-176.404,7.183,148.298
C02715=1212.992,310.304,-68.990,-176.402,7.185,148.298
C02716=1212.987,310.553,-69.020,-176.399,7.188,148.298
C02717=1212.983,310.801,-69.050,-176.397,7.190,148.298
C02718=1212.979,311.049,-69.080,-176.394,7.193,148.298
C02719=1212.974,311.297,-69.110,-176.392,7.196,148.298
C02720=1212.970,311.545,-69.140,-176.390,7.199,148.298
C02721=1212.965,311.793,-69.171,-176.388,7.201,148.298
C02722=1212.962,312.041,-69.201,-176.385,7.204,148.298
C02723=1212.957,312.290,-69.231,-176.383,7.206,148.298
C02724=1212.953,312.538,-69.261,-176.380,7.209,148.298
C02725=1212.949,312.786,-69.292,-176.378,7.212,148.298
C02726=1212.944,313.034,-69.322,-176.376,7.215,148.298
C02727=1212.940,313.282,-69.352,-176.374,7.217,148.298
C02728=1212.937,313.530,-69.383,-176.371,7.220,148.298
C02729=1212.932,313.779,-69.413,-176.369,7.222,148.298
C02730=1212.928,314.026,-69.443,-176.367,7.225,148.298
C02731=1212.923,314.274,-69.474,-176.364,7.228,148.298
C02732=1212.918,314.522,-69.505,-176.362,7.231,148.298
C02733=1212.914,314.798,-69.538,-176.359,7.234,148.298
C02734=1212.909,315.074,-69.572,-176.356,7.237,148.298
C02735=1212.904,315.351,-69.605,-176.354,7.240,148.299
C02736=1212.899,315.626,-69.640,-176.352,7.243,148.299
C02737=1212.896,315.875,-69.670,-176.349,7.245,148.298
C02738=1212.892,316.123,-69.701,-176.347,7.248,148.298
C02739=1212.887,316.371,-69.731,-176.345,7.251,148.298
C02740=1212.883,316.619,-69.761,-176.342,7.254,148.299
C02741=1212.878,316.867,-69.792,-176.340,7.256,148.299
C02742=1212.875,317.115,-69.822,-176.338,7.259,148.299
C02743=1212.870,317.363,-69.853,-176.336,7.261,148.299
C02744=1212.866,317.611,-69.884,-176.333,7.264,148.299
C02745=1212.862,317.859,-69.914,-176.331,7.267,148.299
C02746=1212.858,318.108,-69.945,-176.329,7.270,148.299
C02747=1212.853,318.356,-69.975,-176.326,7.273,148.299
C02748=1212.849,318.604,-70.005,-176.324,7.275,148.299
C02749=1212.844,318.852,-70.036,-176.322,7.279,148.299
C02750=1212.840,319.100,-70.067,-176.319,7.281,148.299
C02751=1212.837,319.348,-70.098,-176.317,7.284,148.299
C02752=1212.832,319.596,-70.128,-176.315,7.286,148.299
C02753=1212.828,319.845,-70.159,-176.312,7.289,148.299
C02754=1212.823,320.093,-70.190,-176.310,7.292,148.299
C02755=1212.819,320.340,-70.220,-176.308,7.295,148.299
C02756=1212.815,320.588,-70.251,-176.306,7.297,148.299
C02757=1212.811,320.837,-70.282,-176.303,7.300,148.299
C02758=1212.806,321.085,-70.313,-176.301,7.302,148.299
C02759=1212.802,321.332,-70.343,-176.299,7.306,148.299
C02760=1212.798,321.581,-70.374,-176.297,7.308,148.299
C02761=1212.794,321.828,-70.406,-176.294,7.311,148.299
C02762=1212.789,322.076,-70.437,-176.293,7.314,148.299
C02763=1212.786,322.325,-70.467,-176.290,7.317,148.299
C02764=1212.781,322.573,-70.498,-176.287,7.320,148.299
C02765=1212.777,322.821,-70.529,-176.286,7.322,148.300
C02766=1212.773,323.069,-70.560,-176.283,7.325,148.300
C02767=1212.768,323.317,-70.591,-176.281,7.327,148.300
C02768=1212.764,323.565,-70.622,-176.279,7.331,148.300
C02769=1212.761,323.813,-70.653,-176.276,7.333,148.300
C02770=1212.756,324.061,-70.683,-176.274,7.336,148.300
C02771=1212.751,324.309,-70.714,-176.272,7.339,148.300
C02772=1212.747,324.558,-70.745,-176.269,7.342,148.300
C02773=1212.743,324.805,-70.777,-176.268,7.344,148.300
C02774=1212.739,325.054,-70.808,-176.265,7.347,148.300
C02775=1212.734,325.302,-70.839,-176.264,7.350,148.300
C02776=1212.731,325.549,-70.869,-176.261,7.353,148.300
C02777=1212.727,325.797,-70.901,-176.258,7.356,148.300
C02778=1212.722,326.045,-70.931,-176.257,7.358,148.300
C02779=1212.718,326.294,-70.962,-176.254,7.361,148.300
C02780=1212.714,326.541,-70.994,-176.252,7.364,148.301
C02781=1212.709,326.789,-71.025,-176.250,7.367,148.301
C02782=1212.705,327.038,-71.056,-176.248,7.369,148.301
C02783=1212.701,327.285,-71.087,-176.245,7.372,148.301
C02784=1212.697,327.534,-71.118,-176.244,7.375,148.301
C02785=1212.692,327.782,-71.149,-176.241,7.378,148.301
C02786=1212.689,328.030,-71.181,-176.239,7.380,148.301
C02787=1212.684,328.278,-71.212,-176.237,7.384,148.301
C02788=1212.679,328.526,-71.243,-176.234,7.386,148.301
C02789=1212.676,328.774,-71.274,-176.232,7.389,148.301
C02790=1212.671,329.022,-71.305,-176.230,7.391,148.301
C02791=1212.667,329.270,-71.337,-176.228,7.395,148.301
C02792=1212.663,329.518,-71.368,-176.225,7.398,148.301
C02793=1212.659,329.766,-71.400,-176.224,7.400,148.302
C02794=1212.655,330.014,-71.430,-176.221,7.403,148.302
C02795=1212.651,330.262,-71.462,-176.219,7.406,148.302
C02796=1212.646,330.510,-71.493,-176.217,7.409,148.302
C02797=1212.642,330.758,-71.525,-176.215,7.411,148.302
C02798=1212.638,331.006,-71.556,-176.213,7.415,148.302
C02799=1212.634,331.254,-71.588,-176.211,7.417,148.302
C02800=1212.630,331.502,-71.618,-176.208,7.420,148.302
C02801=1212.626,331.750,-71.650,-176.206,7.422,148.302
C02802=1212.621,331.998,-71.681,-176.204,7.426,148.303
C02803=1212.617,332.246,-71.713,-176.202,7.428,148.303
C02804=1212.612,332.493,-71.745,-176.200,7.431,148.303
C02805=1212.608,332.742,-71.776,-176.198,7.434,148.303
C02806=1212.604,332.989,-71.807,-176.196,7.437,148.303
C02807=1212.600,333.238,-71.839,-176.193,7.440,148.303
C02808=1212.596,333.485,-71.870,-176.191,7.442,148.303
C02809=1212.592,333.733,-71.902,-176.189,7.446,148.303
C02810=1212.588,333.981,-71.933,-176.187,7.448,148.303
C02811=1212.583,334.230,-71.965,-176.185,7.451,148.303
C02812=1212.579,334.477,-71.997,-176.183,7.454,148.304
C02813=1212.575,334.726,-72.028,-176.180,7.457,148.304
C02814=1212.570,334.973,-72.059,-176.179,7.459,148.304
C02815=1212.567,335.221,-72.091,-176.177,7.463,148.304
C02816=1212.563,335.469,-72.123,-176.174,7.465,148.304
C02817=1212.558,335.717,-72.154,-176.172,7.468,148.304
C02818=1212.554,335.965,-72.186,-176.171,7.471,148.304
C02819=1212.550,336.213,-72.218,-176.168,7.474,148.304
C02820=1212.546,336.461,-72.249,-176.166,7.476,148.305
C02821=1212.541,336.709,-72.281,-176.164,7.480,148.305
C02822=1212.537,336.957,-72.313,-176.162,7.482,148.305
C02823=1212.533,337.205,-72.344,-176.160,7.485,148.305
C02824=1212.529,337.452,-72.376,-176.158,7.489,148.305
C02825=1212.524,337.701,-72.408,-176.156,7.491,148.305
C02826=1212.520,337.948,-72.440,-176.153,7.494,148.305
C02827=1212.516,338.197,-72.471,-176.152,7.497,148.306
C02828=1212.512,338.445,-72.503,-176.149,7.500,148.306
C02829=1212.507,338.692,-72.535,-176.148,7.503,148.306
C02830=1212.504,338.941,-72.567,-176.145,7.506,148.306
C02831=1212.500,339.189,-72.599,-176.143,7.508,148.306
C02832=1212.495,339.436,-72.631,-176.141,7.512,148.306
C02833=1212.491,339.684,-72.662,-176.140,7.514,148.307
C02834=1212.487,339.932,-72.694,-176.137,7.517,148.307
C02835=1212.482,340.180,-72.726,-176.135,7.520,148.307
C02836=1212.479,340.428,-72.758,-176.133,7.523,148.307
C02837=1212.474,340.706,-72.793,-176.131,7.526,148.307
C02838=1212.469,340.984,-72.829,-176.129,7.530,148.307
C02839=1212.464,341.262,-72.866,-176.126,7.533,148.307
C02840=1212.460,341.540,-72.902,-176.124,7.536,148.308
C02841=1212.455,341.788,-72.934,-176.122,7.539,148.308
C02842=1212.452,342.036,-72.965,-176.120,7.542,148.308
C02843=1212.448,342.284,-72.997,-176.118,7.544,148.308
C02844=1212.443,342.531,-73.029,-176.116,7.548,148.309
C02845=1212.439,342.779,-73.061,-176.114,7.550,148.308
C02846=1212.435,343.028,-73.094,-176.112,7.553,148.309
C02847=1212.430,343.275,-73.125,-176.110,7.556,148.309
C02848=1212.426,343.524,-73.158,-176.108,7.559,148.309
C02849=1212.422,343.772,-73.189,-176.106,7.562,148.309
C02850=1212.418,344.019,-73.221,-176.104,7.565,148.309
C02851=1212.413,344.267,-73.253,-176.102,7.568,148.310
C02852=1212.410,344.515,-73.286,-176.100,7.571,148.310
C02853=1212.406,344.763,-73.318,-176.099,7.573,148.310
C02854=1212.401,345.010,-73.350,-176.096,7.577,148.310
C02855=1212.397,345.259,-73.382,-176.094,7.579,148.310
C02856=1212.393,345.507,-73.414,-176.092,7.582,148.310
C02857=1212.389,345.755,-73.447,-176.090,7.585,148.311
C02858=1212.385,346.002,-73.479,-176.088,7.588,148.311
C02859=1212.380,346.250,-73.511,-176.086,7.591,148.311
C02860=1212.377,346.498,-73.543,-176.084,7.594,148.311
C02861=1212.372,346.747,-73.575,-176.083,7.597,148.311
C02862=1212.368,346.993,-73.608,-176.080,7.600,148.312
C02863=1212.364,347.242,-73.640,-176.079,7.602,148.312
C02864=1212.359,347.490,-73.673,-176.077,7.606,148.312
C02865=1212.356,347.737,-73.705,-176.075,7.608,148.312
C02866=1212.351,347.985,-73.737,-176.073,7.612,148.313
C02867=1212.347,348.233,-73.769,-176.071,7.614,148.313
C02868=1212.343,348.481,-73.801,-176.069,7.618,148.313
C02869=1212.339,348.729,-73.834,-176.067,7.620,148.313
C02870=1212.335,348.977,-73.866,-176.065,7.623,148.313
C02871=1212.330,349.224,-73.899,-176.063,7.626,148.314
C02872=1212.326,349.472,-73.931,-176.062,7.629,148.314
C02873=1212.322,349.721,-73.964,-176.060,7.632,148.314
C02874=1212.318,349.968,-73.996,-176.058,7.635,148.314
C02875=1212.314,350.216,-74.029,-176.056,7.638,148.315
C02876=1212.309,350.464,-74.061,-176.054,7.641,148.315
C02877=1212.306,350.711,-74.093,-176.052,7.644,148.315
C02878=1212.301,350.960,-74.126,-176.051,7.646,148.315
C02879=1212.297,351.208,-74.159,-176.048,7.650,148.315
C02880=1212.293,351.456,-74.191,-176.047,7.652,148.316
C02881=1212.289,351.703,-74.224,-176.045,7.656,148.316
C02882=1212.284,351.951,-74.256,-176.043,7.658,148.316
C02883=1212.281,352.198,-74.288,-176.041,7.662,148.316
C02884=1212.276,352.447,-74.321,-176.040,7.664,148.317
C02885=1212.272,352.694,-74.354,-176.037,7.668,148.317
C02886=1212.268,352.942,-74.386,-176.036,7.670,148.317
C02887=1212.264,353.190,-74.419,-176.034,7.674,148.317
C02888=1212.260,353.439,-74.451,-176.032,7.676,148.318
C02889=1212.255,353.686,-74.484,-176.031,7.679,148.318
C02890=1212.252,353.933,-74.517,-176.028,7.682,148.318
C02891=1212.247,354.181,-74.549,-176.027,7.685,148.318
C02892=1212.243,354.429,-74.582,-176.025,7.688,148.319
C02893=1212.239,354.677,-74.615,-176.023,7.691,148.319
C02894=1212.235,354.925,-74.647,-176.021,7.694,148.319
C02895=1212.231,355.173,-74.681,-176.020,7.697,148.319
C02896=1212.227,355.421,-74.713,-176.018,7.700,148.320
C02897=1212.223,355.669,-74.746,-176.016,7.703,148.320
C02898=1212.219,355.916,-74.779,-176.014,7.705,148.320
C02899=1212.214,356.164,-74.811,-176.013,7.709,148.320
C02900=1212.210,356.411,-74.844,-176.011,7.712,148.321
C02901=1212.206,356.659,-74.877,-176.009,7.715,148.321
C02902=1212.201,356.908,-74.910,-176.007,7.717,148.321
C02903=1212.198,357.155,-74.942,-176.005,7.721,148.321
C02904=1212.194,357.403,-74.975,-176.004,7.724,148.322
C02905=1212.189,357.651,-75.008,-176.002,7.727,148.322
C02906=1212.185,357.899,-75.041,-176.000,7.730,148.322
C02907=1212.181,358.146,-75.074,-175.999,7.732,148.322
C02908=1212.177,358.394,-75.107,-175.997,7.736,148.323
C02909=1212.173,358.643,-75.140,-175.995,7.738,148.323
C02910=1212.169,358.890,-75.172,-175.993,7.742,148.323
C02911=1212.165,359.138,-75.205,-175.992,7.745,148.324
C02912=1212.161,359.385,-75.238,-175.990,7.747,148.324
C02913=1212.157,359.633,-75.272,-175.989,7.751,148.324
C02914=1212.153,359.881,-75.305,-175.987,7.753,148.325
C02915=1212.148,360.129,-75.337,-175.985,7.757,148.325
C02916=1212.144,360.377,-75.370,-175.984,7.759,148.325
C02917=1212.140,360.625,-75.404,-175.982,7.762,148.325
C02918=1212.136,360.872,-75.437,-175.980,7.766,148.326
C02919=1212.132,361.120,-75.469,-175.979,7.768,148.326
C02920=1212.128,361.368,-75.502,-175.977,7.772,148.326
C02921=1212.124,361.615,-75.536,-175.975,7.774,148.327
C02922=1212.120,361.863,-75.569,-175.974,7.777,148.327
C02923=1212.116,362.111,-75.602,-175.972,7.780,148.327
C02924=1212.111,362.359,-75.634,-175.971,7.783,148.328
C02925=1212.107,362.607,-75.667,-175.969,7.786,148.328
C02926=1212.103,362.855,-75.701,-175.967,7.789,148.328
C02927=1212.099,363.102,-75.734,-175.966,7.792,148.329
C02928=1212.095,363.350,-75.767,-175.964,7.796,148.329
C02929=1212.091,363.598,-75.800,-175.963,7.798,148.329
C02930=1212.087,363.845,-75.833,-175.961,7.801,148.329
C02931=1212.082,364.093,-75.866,-175.959,7.805,148.330
C02932=1212.078,364.341,-75.900,-175.957,7.807,148.330
C02933=1212.074,364.589,-75.933,-175.956,7.810,148.330
C02934=1212.070,364.836,-75.966,-175.955,7.814,148.331
C02935=1212.066,365.084,-75.999,-175.953,7.816,148.331
C02936=1212.062,365.331,-76.033,-175.952,7.819,148.331
C02937=1212.058,365.579,-76.066,-175.951,7.822,148.332
C02938=1212.054,365.827,-76.099,-175.948,7.825,148.332
C02939=1212.050,366.075,-76.133,-175.947,7.828,148.332
C02940=1212.046,366.323,-76.166,-175.946,7.831,148.333
C02941=1212.041,366.603,-76.204,-175.944,7.834,148.333
C02942=1212.036,366.884,-76.241,-175.942,7.838,148.334
C02943=1212.032,367.163,-76.279,-175.941,7.841,148.334
C02944=1212.027,367.444,-76.317,-175.939,7.844,148.334
C02945=1212.023,367.692,-76.350,-175.938,7.847,148.335
C02946=1212.019,367.939,-76.384,-175.936,7.851,148.335
C02947=1212.015,368.187,-76.417,-175.934,7.853,148.335
C02948=1212.011,368.435,-76.450,-175.933,7.856,148.336
C02949=1212.007,368.682,-76.484,-175.932,7.859,148.336
C02950=1212.003,368.930,-76.517,-175.930,7.862,148.337
C02951=1211.998,369.177,-76.550,-175.929,7.865,148.337
C02952=1211.994,369.425,-76.583,-175.927,7.868,148.337
C02953=1211.990,369.673,-76.618,-175.926,7.871,148.338
C02954=1211.986,369.921,-76.651,-175.925,7.874,148.338
C02955=1211.982,370.169,-76.684,-175.923,7.877,148.338
C02956=1211.978,370.416,-76.717,-175.922,7.880,148.339
C02957=1211.974,370.663,-76.751,-175.921,7.883,148.339
C02958=1211.970,370.911,-76.784,-175.920,7.885,148.340
C02959=1211.965,371.159,-76.818,-175.918,7.888,148.340
C02960=1211.961,371.408,-76.852,-175.916,7.892,148.340
C02961=1211.958,371.655,-76.886,-175.915,7.894,148.341
C02962=1211.954,371.903,-76.919,-175.914,7.897,148.341
C02963=1211.949,372.150,-76.952,-175.913,7.900,148.341
C02964=1211.945,372.398,-76.986,-175.912,7.903,148.342
C02965=1211.941,372.645,-77.020,-175.910,7.906,148.342
C02966=1211.937,372.894,-77.053,-175.909,7.909,148.343
C02967=1211.933,373.141,-77.087,-175.907,7.912,148.343
C02968=1211.928,373.389,-77.121,-175.906,7.915,148.343
C02969=1211.925,373.636,-77.155,-175.905,7.918,148.344
C02970=1211.920,373.884,-77.188,-175.904,7.921,148.344
C02971=1211.916,374.132,-77.221,-175.903,7.923,148.345
C02972=1211.912,374.380,-77.256,-175.901,7.926,148.345
C02973=1211.908,374.627,-77.289,-175.900,7.929,148.345
C02974=1211.904,374.875,-77.323,-175.899,7.932,148.346
C02975=1211.900,375.122,-77.356,-175.897,7.936,148.346
C02976=1211.896,375.370,-77.390,-175.896,7.938,148.347
C02977=1211.892,375.618,-77.424,-175.895,7.941,148.347
C02978=1211.888,375.866,-77.457,-175.894,7.944,148.347
C02979=1211.883,376.113,-77.492,-175.892,7.947,148.348
C02980=1211.879,376.361,-77.525,-175.892,7.950,148.348
C02981=1211.876,376.609,-77.559,-175.891,7.953,148.349
C02982=1211.872,376.857,-77.592,-175.889,7.955,148.349
C02983=1211.867,377.104,-77.627,-175.888,7.958,148.350
C02984=1211.863,377.352,-77.660,-175.887,7.961,148.350
C02985=1211.859,377.599,-77.694,-175.886,7.964,148.350
C02986=1211.855,377.847,-77.728,-175.885,7.967,148.351
C02987=1211.851,378.095,-77.762,-175.883,7.970,148.351
C02988=1211.847,378.342,-77.795,-175.883,7.973,148.352
C02989=1211.843,378.590,-77.829,-175.881,7.975,148.352
C02990=1211.839,378.838,-77.863,-175.880,7.978,148.353
C02991=1211.834,379.086,-77.897,-175.879,7.981,148.353
C02992=1211.831,379.333,-77.931,-175.878,7.984,148.353
C02993=1211.827,379.580,-77.965,-175.877,7.987,148.354
C02994=1211.823,379.829,-77.999,-175.876,7.990,148.354
C02995=1211.819,380.076,-78.033,-175.875,7.993,148.355
C02996=1211.814,380.324,-78.067,-175.873,7.995,148.355
C02997=1211.811,380.572,-78.101,-175.873,7.998,148.356
C02998=1211.807,380.819,-78.135,-175.872,8.001,148.356
C02999=1211.802,381.067,-78.169,-175.871,8.003,148.356
C03000=1211.798,381.314,-78.202,-175.870,8.006,148.357
C03001=1211.794,381.562,-78.237,-175.869,8.009,148.357
C03002=1211.790,381.810,-78.270,-175.868,8.012,148.358
C03003=1211.786,382.057,-78.304,-175.867,8.015,148.358
C03004=1211.782,382.304,-78.339,-175.866,8.018,148.359
C03005=1211.778,382.553,-78.372,-175.865,8.021,148.359
C03006=1211.773,382.800,-78.407,-175.864,8.023,148.360
C03007=1211.770,383.047,-78.441,-175.863,8.026,148.360
C03008=1211.765,383.296,-78.475,-175.862,8.029,148.361
C03009=1211.761,383.543,-78.509,-175.861,8.032,148.361
C03010=1211.757,383.790,-78.543,-175.860,8.035,148.362
C03011=1211.754,384.038,-78.577,-175.859,8.037,148.362
C03012=1211.749,384.286,-78.611,-175.858,8.039,148.362
C03013=1211.745,384.533,-78.645,-175.857,8.043,148.363
C03014=1211.741,384.781,-78.680,-175.856,8.045,148.363
C03015=1211.737,385.029,-78.714,-175.855,8.048,148.364
C03016=1211.733,385.276,-78.748,-175.854,8.051,148.364
C03017=1211.729,385.524,-78.782,-175.854,8.053,148.365
C03018=1211.725,385.772,-78.816,-175.853,8.056,148.365
C03019=1211.721,386.019,-78.850,-175.852,8.059,148.366
C03020=1211.717,386.267,-78.885,-175.851,8.062,148.366
C03021=1211.713,386.514,-78.919,-175.850,8.064,148.366
C03022=1211.708,386.762,-78.952,-175.849,8.067,148.367
C03023=1211.705,387.010,-78.987,-175.848,8.070,148.367
C03024=1211.700,387.257,-79.021,-175.847,8.073,148.368
C03025=1211.696,387.505,-79.055,-175.847,8.075,148.368
C03026=1211.692,387.753,-79.090,-175.846,8.078,148.369
C03027=1211.689,388.000,-79.124,-175.845,8.081,148.369
C03028=1211.684,388.247,-79.158,-175.844,8.083,148.370
C03029=1211.680,388.496,-79.192,-175.844,8.086,148.370
C03030=1211.676,388.743,-79.226,-175.842,8.089,148.371
C03031=1211.672,388.991,-79.261,-175.842,8.091,148.371
C03032=1211.668,389.238,-79.295,-175.841,8.094,148.372
C03033=1211.664,389.486,-79.329,-175.840,8.097,148.372
C03034=1211.660,389.734,-79.363,-175.840,8.099,148.373
C03035=1211.656,389.981,-79.398,-175.839,8.102,148.373
C03036=1211.652,390.228,-79.432,-175.838,8.105,148.374
C03037=1211.648,390.476,-79.467,-175.837,8.107,148.374
C03038=1211.643,390.724,-79.501,-175.836,8.110,148.375
C03039=1211.640,390.971,-79.535,-175.835,8.113,148.375
C03040=1211.636,391.219,-79.570,-175.835,8.115,148.375
C03041=1211.632,391.466,-79.604,-175.834,8.118,148.376
C03042=1211.628,391.714,-79.639,-175.833,8.120,148.376
C03043=1211.623,391.961,-79.673,-175.833,8.124,148.377
C03044=1211.620,392.209,-79.707,-175.832,8.126,148.377
C03045=1211.615,392.492,-79.746,-175.831,8.129,148.378
C03046=1211.610,392.774,-79.786,-175.830,8.132,148.378
C03047=1211.605,393.056,-79.825,-175.830,8.135,148.379
C03048=1211.601,393.339,-79.864,-175.829,8.138,148.379
C03049=1211.597,393.586,-79.898,-175.828,8.141,148.380
C03050=1211.593,393.834,-79.933,-175.828,8.143,148.381
C03051=1211.589,394.081,-79.968,-175.826,8.146,148.381
C03052=1211.585,394.328,-80.001,-175.826,8.148,148.382
C03053=1211.581,394.576,-80.036,-175.825,8.151,148.382
C03054=1211.576,394.824,-80.071,-175.825,8.153,148.382
C03055=1211.573,395.072,-80.105,-175.824,8.156,148.383
C03056=1211.568,395.319,-80.139,-175.823,8.158,148.383
C03057=1211.565,395.567,-80.174,-175.823,8.161,148.384
C03058=1211.561,395.814,-80.208,-175.822,8.163,148.384
C03059=1211.556,396.061,-80.243,-175.822,8.166,148.385
C03060=1211.552,396.309,-80.278,-175.821,8.168,148.385
C03061=1211.549,396.556,-80.312,-175.820,8.171,148.386
C03062=1211.545,396.804,-80.347,-175.820,8.174,148.386
C03063=1211.540,397.052,-80.381,-175.819,8.176,148.387
C03064=1211.536,397.300,-80.416,-175.818,8.179,148.387
C03065=1211.532,397.547,-80.450,-175.818,8.181,148.388
C03066=1211.528,397.795,-80.485,-175.817,8.183,148.388
C03067=1211.524,398.042,-80.520,-175.817,8.186,148.389
C03068=1211.520,398.290,-80.555,-175.816,8.188,148.389
C03069=1211.516,398.537,-80.589,-175.816,8.190,148.390
C03070=1211.512,398.785,-80.623,-175.815,8.194,148.390
C03071=1211.508,399.033,-80.658,-175.814,8.196,148.391
C03072=1211.504,399.280,-80.692,-175.814,8.199,148.391
C03073=1211.500,399.527,-80.727,-175.813,8.201,148.392
C03074=1211.496,399.775,-80.762,-175.813,8.203,148.392
C03075=1211.492,400.023,-80.797,-175.812,8.206,148.393
C03076=1211.487,400.270,-80.831,-175.811,8.208,148.393
C03077=1211.484,400.518,-80.865,-175.811,8.210,148.394
C03078=1211.480,400.765,-80.901,-175.810,8.213,148.394
C03079=1211.476,401.013,-80.935,-175.810,8.215,148.394
C03080=1211.471,401.260,-80.970,-175.809,8.218,148.395
C03081=1211.468,401.508,-81.004,-175.809,8.220,148.396
C03082=1211.464,401.755,-81.039,-175.808,8.223,148.396
C03083=1211.460,402.003,-81.074,-175.808,8.225,148.396
C03084=1211.455,402.251,-81.109,-175.807,8.227,148.397
C03085=1211.451,402.499,-81.143,-175.806,8.230,148.397
C03086=1211.448,402.745,-81.178,-175.806,8.232,148.398
C03087=1211.444,402.993,-81.213,-175.806,8.234,148.398
C03088=1211.439,403.241,-81.247,-175.805,8.237,148.399
C03089=1211.435,403.489,-81.282,-175.805,8.240,148.399
C03090=1211.431,403.736,-81.317,-175.804,8.242,148.400
C03091=1211.428,403.984,-81.352,-175.804,8.244,148.400
C03092=1211.423,404.231,-81.386,-175.804,8.246,148.401
C03093=1211.419,404.478,-81.422,-175.802,8.249,148.401
C03094=1211.415,404.726,-81.456,-175.802,8.251,148.402
C03095=1211.411,404.974,-81.491,-175.802,8.254,148.402
C03096=1211.407,405.221,-81.526,-175.801,8.256,148.403
C03097=1211.403,405.469,-81.560,-175.801,8.258,148.403
C03098=1211.399,405.717,-81.595,-175.800,8.261,148.404
C03099=1211.395,405.963,-81.630,-175.800,8.263,148.404
C03100=1211.391,406.212,-81.665,-175.799,8.265,148.405
C03101=1211.386,406.459,-81.700,-175.799,8.267,148.405
C03102=1211.383,406.707,-81.735,-175.799,8.269,148.406
C03103=1211.379,406.954,-81.769,-175.798,8.272,148.406
C03104=1211.375,407.202,-81.804,-175.797,8.274,148.406
C03105=1211.371,407.449,-81.839,-175.797,8.277,148.407
C03106=1211.367,407.697,-81.874,-175.797,8.279,148.408
C03107=1211.363,407.943,-81.909,-175.796,8.281,148.408
C03108=1211.359,408.192,-81.944,-175.796,8.283,148.408
C03109=1211.355,408.440,-81.979,-175.796,8.285,148.409
C03110=1211.350,408.687,-82.014,-175.795,8.287,148.409
C03111=1211.347,408.934,-82.048,-175.795,8.290,148.410
C03112=1211.343,409.181,-82.083,-175.794,8.293,148.410
C03113=1211.339,409.429,-82.118,-175.793,8.295,148.411
C03114=1211.335,409.676,-82.153,-175.793,8.297,148.411
C03115=1211.331,409.924,-82.188,-175.792,8.299,148.412
C03116=1211.326,410.172,-82.223,-175.792,8.301,148.412
C03117=1211.322,410.419,-82.258,-175.792,8.304,148.413
C03118=1211.318,410.667,-82.293,-175.791,8.306,148.413
C03119=1211.314,410.914,-82.328,-175.791,8.308,148.414
C03120=1211.310,411.162,-82.363,-175.791,8.310,148.414
C03121=1211.307,411.409,-82.398,-175.790,8.312,148.414
C03122=1211.303,411.657,-82.432,-175.790,8.314,148.415
C03123=1211.299,411.904,-82.468,-175.789,8.316,148.415
C03124=1211.294,412.152,-82.502,-175.789,8.319,148.416
C03125=1211.291,412.399,-82.538,-175.788,8.322,148.416
C03126=1211.286,412.647,-82.573,-175.788,8.324,148.417
C03127=1211.283,412.894,-82.608,-175.788,8.326,148.417
C03128=1211.278,413.142,-82.643,-175.787,8.328,148.418
C03129=1211.274,413.389,-82.678,-175.787,8.330,148.418
C03130=1211.270,413.637,-82.713,-175.787,8.332,148.419
C03131=1211.266,413.884,-82.748,-175.786,8.334,148.419
C03132=1211.262,414.132,-82.783,-175.786,8.337,148.420
C03133=1211.258,414.379,-82.818,-175.785,8.339,148.420
C03134=1211.254,414.627,-82.853,-175.785,8.341,148.420
C03135=1211.250,414.874,-82.888,-175.785,8.343,148.421
C03136=1211.246,415.122,-82.923,-175.784,8.345,148.421
C03137=1211.242,415.368,-82.958,-175.784,8.347,148.422
C03138=1211.238,415.615,-82.993,-175.783,8.349,148.422
C03139=1211.234,415.860,-83.028,-175.783,8.352,148.423
C03140=1211.230,416.107,-83.063,-175.782,8.354,148.423
C03141=1211.226,416.354,-83.097,-175.782,8.356,148.424
C03142=1211.222,416.600,-83.133,-175.782,8.358,148.424
C03143=1211.221,416.846,-83.167,-175.782,8.359,148.424
C03144=1211.222,417.092,-83.201,-175.781,8.361,148.425
C03145=1210.800,417.092,-83.238,-175.784,8.372,148.428
C03146=1210.799,416.845,-83.203,-175.785,8.370,148.428
C03147=1210.800,416.597,-83.168,-175.785,8.369,148.428
C03148=1210.804,416.349,-83.134,-175.785,8.367,148.427
C03149=1210.808,416.101,-83.098,-175.785,8.364,148.427
C03150=1210.812,415.854,-83.064,-175.786,8.362,148.426
C03151=1210.816,415.606,-83.028,-175.786,8.360,148.426
C03152=1210.820,415.358,-82.993,-175.787,8.358,148.425
C03153=1210.824,415.111,-82.958,-175.787,8.356,148.425
C03154=1210.828,414.863,-82.923,-175.787,8.354,148.424
C03155=1210.833,414.617,-82.888,-175.788,8.352,148.424
C03156=1210.837,414.368,-82.853,-175.788,8.349,148.424
C03157=1210.840,414.121,-82.818,-175.789,8.347,148.423
C03158=1210.844,413.874,-82.782,-175.789,8.345,148.423
C03159=1210.848,413.626,-82.748,-175.789,8.343,148.422
C03160=1210.852,413.378,-82.712,-175.790,8.341,148.422
C03161=1210.857,413.131,-82.678,-175.790,8.339,148.421
C03162=1210.860,412.884,-82.642,-175.790,8.336,148.421
C03163=1210.865,412.636,-82.608,-175.791,8.334,148.420
C03164=1210.869,412.389,-82.572,-175.791,8.332,148.420
C03165=1210.873,412.141,-82.538,-175.792,8.330,148.420
C03166=1210.877,411.894,-82.502,-175.793,8.327,148.419
C03167=1210.881,411.646,-82.467,-175.793,8.325,148.418
C03168=1210.885,411.399,-82.432,-175.794,8.323,148.418
C03169=1210.888,411.151,-82.398,-175.794,8.320,148.418
C03170=1210.893,410.904,-82.363,-175.794,8.318,148.417
C03171=1210.897,410.656,-82.328,-175.795,8.316,148.417
C03172=1210.900,410.408,-82.293,-175.795,8.314,148.416
C03173=1210.905,410.161,-82.258,-175.796,8.312,148.416
C03174=1210.909,409.913,-82.223,-175.796,8.310,148.415
C03175=1210.913,409.666,-82.188,-175.796,8.307,148.415
C03176=1210.917,409.418,-82.153,-175.797,8.305,148.414
C03177=1210.921,409.171,-82.118,-175.797,8.303,148.414
C03178=1210.925,408.923,-82.083,-175.797,8.301,148.413
C03179=1210.929,408.676,-82.047,-175.798,8.298,148.413
C03180=1210.933,408.429,-82.013,-175.799,8.296,148.412
C03181=1210.937,408.180,-81.979,-175.799,8.294,148.412
C03182=1210.941,407.934,-81.943,-175.799,8.292,148.412
C03183=1210.945,407.686,-81.909,-175.800,8.289,148.411
C03184=1210.949,407.439,-81.873,-175.800,8.287,148.411
C03185=1210.953,407.191,-81.839,-175.800,8.285,148.410
C03186=1210.958,406.943,-81.804,-175.801,8.283,148.410
C03187=1210.961,406.696,-81.769,-175.801,8.280,148.409
C03188=1210.965,406.448,-81.734,-175.802,8.278,148.409
C03189=1210.969,406.200,-81.700,-175.802,8.275,148.408
C03190=1210.973,405.953,-81.664,-175.803,8.274,148.408
C03191=1210.977,405.706,-81.630,-175.803,8.271,148.407
C03192=1210.981,405.458,-81.594,-175.804,8.268,148.407
C03193=1210.986,405.211,-81.560,-175.805,8.266,148.406
C03194=1210.990,404.963,-81.525,-175.805,8.264,148.406
C03195=1210.993,404.716,-81.490,-175.805,8.262,148.405
C03196=1210.997,404.468,-81.456,-175.806,8.260,148.405
C03197=1211.002,404.220,-81.421,-175.806,8.257,148.404
C03198=1211.005,403.973,-81.386,-175.807,8.254,148.404
C03199=1211.010,403.726,-81.351,-175.807,8.252,148.404
C03200=1211.013,403.478,-81.317,-175.807,8.250,148.403
C03201=1211.018,403.230,-81.282,-175.808,8.248,148.402
C03202=1211.021,402.983,-81.247,-175.809,8.245,148.402
C03203=1211.026,402.735,-81.212,-175.809,8.243,148.401
C03204=1211.030,402.487,-81.178,-175.809,8.240,148.401
C03205=1211.034,402.240,-81.142,-175.810,8.238,148.401
C03206=1211.037,401.993,-81.108,-175.811,8.235,148.400
C03207=1211.041,401.745,-81.073,-175.811,8.233,148.399
C03208=1211.046,401.497,-81.039,-175.812,8.231,148.399
C03209=1211.050,401.250,-81.003,-175.812,8.228,148.399
C03210=1211.053,401.003,-80.969,-175.813,8.226,148.398
C03211=1211.057,400.754,-80.935,-175.813,8.224,148.398
C03212=1211.062,400.507,-80.900,-175.814,8.221,148.397
C03213=1211.066,400.260,-80.865,-175.815,8.219,148.397
C03214=1211.070,400.012,-80.830,-175.815,8.216,148.396
C03215=1211.074,399.765,-80.796,-175.816,8.213,148.396
C03216=1211.078,399.517,-80.761,-175.816,8.211,148.395
C03217=1211.083,399.269,-80.727,-175.816,8.209,148.395
C03218=1211.086,399.022,-80.691,-175.817,8.206,148.394
C03219=1211.090,398.775,-80.658,-175.818,8.204,148.394
C03220=1211.094,398.527,-80.623,-175.818,8.202,148.393
C03221=1211.099,398.279,-80.588,-175.819,8.199,148.393
C03222=1211.103,398.031,-80.553,-175.819,8.197,148.392
C03223=1211.106,397.784,-80.520,-175.820,8.194,148.392
C03224=1211.110,397.537,-80.484,-175.821,8.192,148.391
C03225=1211.115,397.289,-80.449,-175.821,8.189,148.391
C03226=1211.119,397.041,-80.415,-175.822,8.186,148.390
C03227=1211.122,396.794,-80.381,-175.823,8.184,148.390
C03228=1211.126,396.546,-80.346,-175.823,8.181,148.389
C03229=1211.131,396.298,-80.311,-175.823,8.179,148.389
C03230=1211.135,396.051,-80.278,-175.824,8.177,148.388
C03231=1211.138,395.804,-80.242,-175.825,8.174,148.388
C03232=1211.143,395.556,-80.208,-175.826,8.172,148.388
C03233=1211.146,395.309,-80.173,-175.826,8.169,148.387
C03234=1211.151,395.061,-80.139,-175.826,8.166,148.386
C03235=1211.155,394.813,-80.104,-175.828,8.164,148.386
C03236=1211.159,394.566,-80.070,-175.828,8.161,148.385
C03237=1211.163,394.318,-80.035,-175.829,8.158,148.385
C03238=1211.167,394.070,-80.001,-175.829,8.156,148.385
C03239=1211.171,393.823,-79.967,-175.830,8.153,148.384
C03240=1211.175,393.575,-79.932,-175.831,8.151,148.384
C03241=1211.180,393.328,-79.898,-175.831,8.148,148.383
C03242=1211.184,393.045,-79.858,-175.832,8.145,148.382
C03243=1211.189,392.763,-79.819,-175.833,8.142,148.382
C03244=1211.193,392.481,-79.780,-175.834,8.140,148.382
C03245=1211.198,392.199,-79.741,-175.834,8.137,148.381
C03246=1211.202,391.951,-79.706,-175.836,8.134,148.381
C03247=1211.206,391.703,-79.672,-175.836,8.132,148.380
C03248=1211.209,391.455,-79.638,-175.837,8.129,148.379
C03249=1211.214,391.208,-79.603,-175.838,8.126,148.379
C03250=1211.218,390.961,-79.569,-175.838,8.123,148.378
C03251=1211.222,390.713,-79.535,-175.839,8.121,148.378
C03252=1211.226,390.465,-79.500,-175.839,8.118,148.378
C03253=1211.230,390.218,-79.466,-175.841,8.116,148.377
C03254=1211.234,389.970,-79.431,-175.841,8.112,148.377
C03255=1211.238,389.723,-79.397,-175.842,8.110,148.376
C03256=1211.242,389.475,-79.363,-175.843,8.107,148.376
C03257=1211.247,389.227,-79.328,-175.844,8.105,148.375
C03258=1211.250,388.980,-79.294,-175.844,8.102,148.375
C03259=1211.254,388.732,-79.259,-175.845,8.099,148.374
C03260=1211.258,388.485,-79.226,-175.846,8.096,148.374
C03261=1211.262,388.237,-79.191,-175.847,8.094,148.373
C03262=1211.266,387.990,-79.157,-175.847,8.091,148.373
C03263=1211.271,387.742,-79.123,-175.849,8.088,148.372
C03264=1211.274,387.494,-79.089,-175.849,8.086,148.372
C03265=1211.279,387.247,-79.054,-175.850,8.083,148.371
C03266=1211.283,386.999,-79.020,-175.851,8.080,148.371
C03267=1211.287,386.751,-78.986,-175.852,8.077,148.370
C03268=1211.291,386.504,-78.951,-175.853,8.075,148.370
C03269=1211.294,386.256,-78.917,-175.853,8.072,148.369
C03270=1211.299,386.008,-78.883,-175.855,8.070,148.369
C03271=1211.303,385.761,-78.849,-175.855,8.066,148.368
C03272=1211.307,385.513,-78.815,-175.856,8.064,148.368
C03273=1211.311,385.266,-78.781,-175.857,8.061,148.368
C03274=1211.315,385.018,-78.746,-175.858,8.059,148.367
C03275=1211.319,384.770,-78.713,-175.859,8.056,148.367
C03276=1211.323,384.523,-78.678,-175.860,8.053,148.366
C03277=1211.327,384.275,-78.644,-175.861,8.051,148.366
C03278=1211.331,384.027,-78.610,-175.861,8.048,148.365
C03279=1211.335,383.780,-78.576,-175.863,8.045,148.365
C03280=1211.340,383.532,-78.542,-175.864,8.042,148.364
C03281=1211.344,383.285,-78.508,-175.864,8.039,148.364
C03282=1211.348,383.037,-78.473,-175.866,8.036,148.363
C03283=1211.352,382.789,-78.440,-175.866,8.034,148.363
C03284=1211.356,382.542,-78.406,-175.867,8.031,148.363
C03285=1211.360,382.294,-78.371,-175.868,8.028,148.362
C03286=1211.364,382.047,-78.337,-175.869,8.025,148.362
C03287=1211.368,381.799,-78.304,-175.870,8.022,148.361
C03288=1211.372,381.551,-78.269,-175.871,8.019,148.361
C03289=1211.376,381.304,-78.235,-175.873,8.017,148.360
C03290=1211.380,381.056,-78.202,-175.874,8.014,148.360
C03291=1211.385,380.808,-78.167,-175.874,8.011,148.359
C03292=1211.388,380.561,-78.133,-175.875,8.009,148.359
C03293=1211.392,380.313,-78.100,-175.876,8.006,148.359
C03294=1211.397,380.065,-78.066,-175.877,8.003,148.358
C03295=1211.400,379.818,-78.031,-175.878,8.000,148.358
C03296=1211.405,379.570,-77.998,-175.880,7.997,148.357
C03297=1211.409,379.323,-77.964,-175.881,7.994,148.357
C03298=1211.413,379.075,-77.931,-175.882,7.991,148.356
C03299=1211.417,378.827,-77.896,-175.883,7.988,148.356
C03300=1211.421,378.580,-77.862,-175.884,7.986,148.356
C03301=1211.425,378.332,-77.829,-175.885,7.983,148.355
C03302=1211.429,378.084,-77.794,-175.886,7.980,148.355
C03303=1211.433,377.836,-77.761,-175.888,7.977,148.354
C03304=1211.437,377.589,-77.727,-175.888,7.974,148.354
C03305=1211.442,377.341,-77.693,-175.889,7.971,148.353
C03306=1211.446,377.094,-77.659,-175.891,7.968,148.353
C03307=1211.450,376.845,-77.625,-175.892,7.966,148.353
C03308=1211.454,376.598,-77.591,-175.893,7.963,148.352
C03309=1211.458,376.350,-77.558,-175.894,7.960,148.352
C03310=1211.462,376.103,-77.524,-175.895,7.957,148.351
C03311=1211.467,375.855,-77.490,-175.897,7.954,148.351
C03312=1211.470,375.607,-77.456,-175.897,7.951,148.350
C03313=1211.474,375.359,-77.423,-175.899,7.948,148.350
C03314=1211.478,375.112,-77.389,-175.900,7.946,148.350
C03315=1211.483,374.864,-77.355,-175.902,7.942,148.349
C03316=1211.486,374.617,-77.322,-175.903,7.939,148.349
C03317=1211.490,374.369,-77.288,-175.904,7.936,148.348
C03318=1211.495,374.121,-77.254,-175.905,7.933,148.348
C03319=1211.499,373.874,-77.220,-175.906,7.931,148.348
C03320=1211.503,373.626,-77.187,-175.908,7.928,148.347
C03321=1211.507,373.379,-77.153,-175.909,7.925,148.347
C03322=1211.511,373.130,-77.119,-175.910,7.922,148.346
C03323=1211.515,372.882,-77.086,-175.911,7.919,148.346
C03324=1211.519,372.635,-77.052,-175.913,7.916,148.346
C03325=1211.523,372.387,-77.019,-175.914,7.913,148.345
C03326=1211.528,372.140,-76.985,-175.915,7.910,148.345
C03327=1211.532,371.892,-76.951,-175.916,7.907,148.344
C03328=1211.535,371.644,-76.918,-175.918,7.905,148.344
C03329=1211.539,371.397,-76.884,-175.919,7.902,148.344
C03330=1211.543,371.149,-76.851,-175.921,7.898,148.343
C03331=1211.548,370.901,-76.817,-175.922,7.896,148.343
C03332=1211.552,370.653,-76.784,-175.923,7.893,148.343
C03333=1211.556,370.406,-76.750,-175.925,7.890,148.342
C03334=1211.560,370.158,-76.717,-175.926,7.887,148.342
C03335=1211.564,369.910,-76.683,-175.928,7.883,148.341
C03336=1211.568,369.663,-76.649,-175.929,7.881,148.341
C03337=1211.572,369.415,-76.616,-175.930,7.878,148.341
C03338=1211.577,369.167,-76.583,-175.932,7.875,148.340
C03339=1211.581,368.919,-76.550,-175.933,7.872,148.340
C03340=1211.585,368.672,-76.516,-175.935,7.869,148.340
C03341=1211.589,368.425,-76.482,-175.936,7.866,148.339
C03342=1211.592,368.176,-76.449,-175.937,7.863,148.339
C03343=1211.596,367.928,-76.416,-175.939,7.860,148.339
C03344=1211.601,367.680,-76.382,-175.940,7.857,148.338
C03345=1211.605,367.433,-76.349,-175.942,7.854,148.338
C03346=1211.610,367.153,-76.311,-175.943,7.851,148.337
C03347=1211.614,366.873,-76.273,-175.945,7.848,148.337
C03348=1211.619,366.593,-76.235,-175.947,7.844,148.337
C03349=1211.624,366.312,-76.198,-175.948,7.841,148.336
C03350=1211.628,366.064,-76.165,-175.950,7.838,148.336
C03351=1211.632,365.816,-76.132,-175.951,7.835,148.335
C03352=1211.636,365.569,-76.098,-175.953,7.832,148.335
C03353=1211.640,365.322,-76.065,-175.954,7.829,148.335
C03354=1211.644,365.074,-76.032,-175.955,7.826,148.334
C03355=1211.648,364.826,-75.999,-175.958,7.823,148.334
C03356=1211.652,364.578,-75.965,-175.959,7.820,148.334
C03357=1211.656,364.331,-75.932,-175.960,7.817,148.333
C03358=1211.660,364.082,-75.899,-175.962,7.814,148.333
C03359=1211.664,363.835,-75.866,-175.963,7.811,148.333
C03360=1211.668,363.587,-75.832,-175.965,7.809,148.333
C03361=1211.672,363.339,-75.799,-175.967,7.805,148.332
C03362=1211.677,363.091,-75.766,-175.968,7.802,148.332
C03363=1211.681,362.844,-75.733,-175.970,7.799,148.332
C03364=1211.685,362.596,-75.700,-175.971,7.796,148.331
C03365=1211.689,362.348,-75.667,-175.973,7.793,148.331
C03366=1211.693,362.100,-75.633,-175.975,7.790,148.331
C03367=1211.697,361.853,-75.600,-175.977,7.787,148.330
C03368=1211.701,361.605,-75.567,-175.978,7.784,148.330
C03369=1211.705,361.357,-75.534,-175.980,7.781,148.330
C03370=1211.710,361.110,-75.501,-175.981,7.778,148.329
C03371=1211.714,360.861,-75.468,-175.983,7.775,148.329
C03372=1211.718,360.613,-75.435,-175.985,7.772,148.329
C03373=1211.722,360.366,-75.402,-175.986,7.770,148.329
C03374=1211.726,360.118,-75.369,-175.988,7.766,148.328
C03375=1211.731,359.870,-75.336,-175.990,7.763,148.328
C03376=1211.734,359.623,-75.303,-175.991,7.760,148.327
C03377=1211.738,359.375,-75.270,-175.993,7.757,148.327
C03378=1211.743,359.127,-75.238,-175.995,7.755,148.327
C03379=1211.747,358.879,-75.204,-175.996,7.751,148.327
C03380=1211.751,358.631,-75.171,-175.998,7.749,148.326
C03381=1211.755,358.384,-75.138,-176.000,7.745,148.326
C03382=1211.759,358.136,-75.105,-176.001,7.742,148.326
C03383=1211.763,357.888,-75.073,-176.004,7.739,148.326
C03384=1211.767,357.640,-75.040,-176.005,7.736,148.325
C03385=1211.771,357.392,-75.007,-176.006,7.734,148.325
C03386=1211.775,357.145,-74.974,-176.009,7.730,148.325
C03387=1211.780,356.897,-74.942,-176.010,7.728,148.324
C03388=1211.784,356.649,-74.908,-176.012,7.724,148.324
C03389=1211.788,356.402,-74.876,-176.014,7.722,148.324
C03390=1211.792,356.154,-74.843,-176.015,7.718,148.324
C03391=1211.796,355.906,-74.810,-176.017,7.716,148.323
C03392=1211.801,355.658,-74.777,-176.019,7.713,148.323
C03393=1211.805,355.410,-74.745,-176.021,7.710,148.323
C03394=1211.808,355.162,-74.712,-176.022,7.707,148.323
C03395=1211.813,354.915,-74.679,-176.024,7.703,148.322
C03396=1211.817,354.666,-74.647,-176.026,7.701,148.322
C03397=1211.821,354.418,-74.613,-176.028,7.697,148.322
C03398=1211.825,354.172,-74.581,-176.029,7.695,148.322
C03399=1211.830,353.923,-74.549,-176.032,7.691,148.321
C03400=1211.834,353.676,-74.516,-176.033,7.689,148.321
C03401=1211.838,353.427,-74.483,-176.035,7.686,148.321
C03402=1211.842,353.180,-74.451,-176.037,7.683,148.321
C03403=1211.846,352.932,-74.418,-176.039,7.679,148.320
C03404=1211.850,352.684,-74.385,-176.040,7.677,148.320
C03405=1211.855,352.435,-74.353,-176.042,7.674,148.320
C03406=1211.859,352.189,-74.320,-176.044,7.671,148.320
C03407=1211.863,351.940,-74.288,-176.046,7.669,148.320
C03408=1211.867,351.693,-74.255,-176.048,7.665,148.319
C03409=1211.871,351.445,-74.223,-176.049,7.662,148.319
C03410=1211.875,351.197,-74.190,-176.052,7.659,148.319
C03411=1211.879,350.949,-74.157,-176.053,7.656,148.318
C03412=1211.883,350.701,-74.125,-176.055,7.653,148.318
C03413=1211.888,350.453,-74.093,-176.057,7.651,148.318
C03414=1211.892,350.206,-74.060,-176.059,7.647,148.318
C03415=1211.896,349.958,-74.028,-176.061,7.645,148.318
C03416=1211.900,349.710,-73.995,-176.063,7.641,148.317
C03417=1211.904,349.462,-73.963,-176.064,7.639,148.317
C03418=1211.909,349.214,-73.931,-176.067,7.635,148.317
C03419=1211.913,348.967,-73.897,-176.068,7.633,148.317
C03420=1211.917,348.719,-73.866,-176.070,7.629,148.316
C03421=1211.921,348.470,-73.833,-176.072,7.627,148.316
C03422=1211.924,348.223,-73.801,-176.074,7.624,148.316
C03423=1211.929,347.975,-73.769,-176.076,7.621,148.316
C03424=1211.934,347.727,-73.736,-176.078,7.618,148.316
C03425=1211.937,347.479,-73.704,-176.080,7.615,148.315
C03426=1211.942,347.231,-73.671,-176.082,7.612,148.315
C03427=1211.946,346.984,-73.640,-176.084,7.609,148.315
C03428=1211.950,346.736,-73.606,-176.086,7.606,148.315
C03429=1211.954,346.488,-73.575,-176.087,7.603,148.315
C03430=1211.958,346.240,-73.542,-176.090,7.600,148.314
C03431=1211.962,345.992,-73.510,-176.091,7.598,148.314
C03432=1211.967,345.744,-73.478,-176.094,7.594,148.314
C03433=1211.970,345.496,-73.446,-176.095,7.592,148.314
C03434=1211.975,345.248,-73.413,-176.097,7.588,148.314
C03435=1211.979,345.001,-73.382,-176.099,7.586,148.313
C03436=1211.984,344.752,-73.349,-176.101,7.582,148.313
C03437=1211.987,344.504,-73.317,-176.103,7.580,148.313
C03438=1211.991,344.257,-73.284,-176.106,7.577,148.313
C03439=1211.996,344.009,-73.253,-176.107,7.574,148.313
C03440=1212.000,343.761,-73.220,-176.109,7.571,148.313
C03441=1212.004,343.513,-73.189,-176.111,7.569,148.312
C03442=1212.009,343.265,-73.156,-176.113,7.565,148.312
C03443=1212.013,343.017,-73.125,-176.115,7.563,148.312
C03444=1212.017,342.769,-73.092,-176.117,7.559,148.312
C03445=1212.021,342.521,-73.060,-176.119,7.557,148.312
C03446=1212.025,342.273,-73.029,-176.121,7.553,148.311
C03447=1212.029,342.026,-72.996,-176.123,7.551,148.311
C03448=1212.033,341.778,-72.964,-176.125,7.548,148.311
C03449=1212.038,341.530,-72.932,-176.127,7.545,148.311
C03450=1212.043,341.252,-72.897,-176.129,7.542,148.311
C03451=1212.047,340.973,-72.860,-176.131,7.539,148.311
C03452=1212.051,340.696,-72.825,-176.134,7.536,148.311
C03453=1212.057,340.417,-72.789,-176.136,7.532,148.310
C03454=1212.060,340.169,-72.757,-176.138,7.529,148.310
C03455=1212.066,339.922,-72.725,-176.140,7.526,148.310
C03456=1212.069,339.674,-72.693,-176.142,7.523,148.310
C03457=1212.073,339.426,-72.662,-176.144,7.521,148.310
C03458=1212.078,339.178,-72.630,-176.147,7.517,148.310
C03459=1212.082,338.930,-72.598,-176.148,7.515,148.309
C03460=1212.085,338.682,-72.566,-176.150,7.512,148.309
C03461=1212.090,338.434,-72.534,-176.153,7.509,148.309
C03462=1212.094,338.186,-72.502,-176.155,7.506,148.309
C03463=1212.098,337.938,-72.470,-176.156,7.504,148.309
C03464=1212.102,337.690,-72.439,-176.159,7.500,148.309
C03465=1212.107,337.442,-72.407,-176.161,7.498,148.309
C03466=1212.111,337.195,-72.375,-176.163,7.495,148.308
C03467=1212.115,336.946,-72.344,-176.165,7.491,148.308
C03468=1212.119,336.698,-72.312,-176.167,7.489,148.308
C03469=1212.124,336.451,-72.280,-176.169,7.486,148.308
C03470=1212.128,336.202,-72.249,-176.171,7.483,148.308
C03471=1212.132,335.955,-72.217,-176.174,7.480,148.308
C03472=1212.136,335.707,-72.185,-176.175,7.478,148.308
C03473=1212.140,335.459,-72.154,-176.178,7.474,148.307
C03474=1212.145,335.210,-72.122,-176.180,7.472,148.307
C03475=1212.148,334.962,-72.090,-176.182,7.469,148.307
C03476=1212.153,334.715,-72.059,-176.184,7.466,148.307
C03477=1212.156,334.467,-72.027,-176.186,7.463,148.307
C03478=1212.161,334.219,-71.996,-176.188,7.461,148.307
C03479=1212.166,333.971,-71.964,-176.190,7.457,148.307
C03480=1212.170,333.723,-71.932,-176.193,7.454,148.307
C03481=1212.174,333.475,-71.901,-176.194,7.452,148.306
C03482=1212.178,333.227,-71.870,-176.197,7.448,148.306
C03483=1212.182,332.979,-71.838,-176.199,7.446,148.306
C03484=1212.186,332.731,-71.807,-176.201,7.443,148.306
C03485=1212.190,332.483,-71.775,-176.203,7.441,148.306
C03486=1212.196,332.235,-71.744,-176.205,7.437,148.306
C03487=1212.199,331.987,-71.712,-176.207,7.435,148.306
C03488=1212.203,331.739,-71.680,-176.210,7.432,148.306
C03489=1212.208,331.491,-71.649,-176.211,7.429,148.305
C03490=1212.212,331.244,-71.618,-176.214,7.426,148.305
C03491=1212.216,330.995,-71.587,-176.216,7.424,148.305
C03492=1212.220,330.748,-71.555,-176.218,7.421,148.305
C03493=1212.224,330.499,-71.524,-176.220,7.417,148.305
C03494=1212.229,330.252,-71.493,-176.223,7.415,148.305
C03495=1212.233,330.003,-71.461,-176.225,7.412,148.305
C03496=1212.237,329.756,-71.430,-176.227,7.409,148.305
C03497=1212.241,329.507,-71.399,-176.229,7.406,148.305
C03498=1212.245,329.260,-71.367,-176.231,7.404,148.305
C03499=1212.249,329.011,-71.336,-176.233,7.401,148.305
C03500=1212.253,328.764,-71.305,-176.236,7.398,148.305
C03501=1212.257,328.515,-71.274,-176.238,7.395,148.304
C03502=1212.262,328.267,-71.243,-176.240,7.393,148.304
C03503=1212.266,328.019,-71.211,-176.242,7.389,148.304
C03504=1212.270,327.771,-71.180,-176.244,7.387,148.304
C03505=1212.275,327.524,-71.149,-176.246,7.384,148.304
C03506=1212.279,327.275,-71.118,-176.249,7.381,148.304
C03507=1212.283,327.027,-71.087,-176.251,7.378,148.304
C03508=1212.287,326.779,-71.055,-176.253,7.375,148.304
C03509=1212.292,326.531,-71.024,-176.255,7.373,148.304
C03510=1212.296,326.283,-70.993,-176.258,7.370,148.304
C03511=1212.300,326.035,-70.962,-176.260,7.368,148.304
C03512=1212.305,325.787,-70.931,-176.262,7.364,148.304
C03513=1212.309,325.539,-70.900,-176.264,7.362,148.304
C03514=1212.313,325.291,-70.869,-176.266,7.359,148.303
C03515=1212.317,325.044,-70.838,-176.268,7.356,148.303
C03516=1212.321,324.795,-70.807,-176.271,7.353,148.303
C03517=1212.325,324.547,-70.776,-176.273,7.350,148.303
C03518=1212.329,324.298,-70.745,-176.275,7.348,148.303
C03519=1212.334,324.051,-70.714,-176.278,7.344,148.303
C03520=1212.338,323.803,-70.683,-176.280,7.342,148.303
C03521=1212.342,323.554,-70.652,-176.282,7.339,148.303
C03522=1212.346,323.307,-70.622,-176.284,7.337,148.303
C03523=1212.351,323.059,-70.591,-176.287,7.334,148.303
C03524=1212.355,322.811,-70.559,-176.288,7.331,148.303
C03525=1212.359,322.563,-70.528,-176.291,7.328,148.303
C03526=1212.364,322.315,-70.497,-176.293,7.326,148.303
C03527=1212.368,322.066,-70.466,-176.295,7.323,148.303
C03528=1212.372,321.818,-70.436,-176.297,7.320,148.303
C03529=1212.376,321.571,-70.405,-176.300,7.317,148.303
C03530=1212.380,321.322,-70.374,-176.302,7.314,148.302
C03531=1212.385,321.074,-70.343,-176.304,7.312,148.302
C03532=1212.389,320.826,-70.313,-176.307,7.309,148.302
C03533=1212.393,320.578,-70.282,-176.309,7.306,148.302
C03534=1212.397,320.330,-70.251,-176.311,7.303,148.302
C03535=1212.402,320.082,-70.220,-176.314,7.301,148.302
C03536=1212.405,319.834,-70.189,-176.316,7.298,148.302
C03537=1212.410,319.586,-70.159,-176.318,7.295,148.302
C03538=1212.414,319.338,-70.128,-176.321,7.292,148.302
C03539=1212.418,319.090,-70.098,-176.323,7.290,148.302
C03540=1212.422,318.841,-70.067,-176.325,7.287,148.302
C03541=1212.427,318.593,-70.036,-176.327,7.285,148.302
C03542=1212.432,318.345,-70.006,-176.330,7.282,148.302
C03543=1212.435,318.097,-69.975,-176.332,7.279,148.302
C03544=1212.440,317.849,-69.944,-176.334,7.276,148.302
C03545=1212.444,317.601,-69.914,-176.337,7.273,148.302
C03546=1212.448,317.353,-69.883,-176.339,7.271,148.302
C03547=1212.452,317.105,-69.852,-176.341,7.268,148.302
C03548=1212.457,316.857,-69.822,-176.343,7.265,148.302
C03549=1212.461,316.609,-69.791,-176.346,7.262,148.302
C03550=1212.465,316.360,-69.761,-176.348,7.260,148.302
C03551=1212.469,316.113,-69.731,-176.351,7.257,148.302
C03552=1212.473,315.864,-69.700,-176.353,7.255,148.302
C03553=1212.478,315.616,-69.669,-176.355,7.251,148.302
C03554=1212.482,315.340,-69.636,-176.358,7.248,148.302
C03555=1212.487,315.064,-69.602,-176.360,7.245,148.302
C03556=1212.492,314.788,-69.568,-176.363,7.242,148.302
C03557=1212.497,314.512,-69.534,-176.366,7.239,148.302
C03558=1212.501,314.264,-69.504,-176.368,7.237,148.302
C03559=1212.505,314.016,-69.473,-176.370,7.234,148.302
C03560=1212.509,313.767,-69.443,-176.372,7.231,148.302
C03561=1212.514,313.520,-69.413,-176.375,7.228,148.302
C03562=1212.518,313.272,-69.383,-176.377,7.226,148.302
C03563=1212.522,313.023,-69.352,-176.379,7.223,148.302
C03564=1212.527,312.775,-69.322,-176.382,7.221,148.302
C03565=1212.531,312.528,-69.292,-176.384,7.218,148.302
C03566=1212.535,312.278,-69.261,-176.386,7.215,148.301
C03567=1212.539,312.031,-69.231,-176.389,7.212,148.301
C03568=1212.544,311.783,-69.200,-176.391,7.210,148.302
C03569=1212.548,311.535,-69.171,-176.393,7.207,148.302
C03570=1212.552,311.287,-69.141,-176.396,7.205,148.302
C03571=1212.557,311.038,-69.111,-176.398,7.202,148.302
C03572=1212.561,310.791,-69.080,-176.400,7.200,148.302
C03573=1212.565,310.543,-69.050,-176.403,7.196,148.301
C03574=1212.569,310.294,-69.020,-176.405,7.194,148.301
C03575=1212.573,310.046,-68.989,-176.407,7.191,148.302
C03576=1212.578,309.798,-68.960,-176.409,7.189,148.302
C03577=1212.582,309.550,-68.929,-176.412,7.186,148.302
C03578=1212.586,309.301,-68.899,-176.414,7.184,148.302
C03579=1212.590,309.054,-68.869,-176.417,7.181,148.302
C03580=1212.595,308.805,-68.839,-176.419,7.178,148.302
C03581=1212.599,308.557,-68.809,-176.422,7.175,148.302
C03582=1212.604,308.309,-68.779,-176.424,7.173,148.302
C03583=1212.608,308.061,-68.749,-176.426,7.170,148.302
C03584=1212.612,307.813,-68.719,-176.429,7.167,148.302
C03585=1212.617,307.564,-68.689,-176.431,7.165,148.302
C03586=1212.621,307.317,-68.659,-176.433,7.162,148.302
C03587=1212.624,307.068,-68.629,-176.436,7.159,148.302
C03588=1212.629,306.820,-68.598,-176.438,7.156,148.302
C03589=1212.633,306.572,-68.569,-176.440,7.154,148.302
C03590=1212.637,306.323,-68.540,-176.443,7.151,148.302
C03591=1212.642,306.075,-68.509,-176.445,7.149,148.302
C03592=1212.646,305.827,-68.479,-176.448,7.146,148.302
C03593=1212.650,305.579,-68.450,-176.450,7.144,148.302
C03594=1212.655,305.331,-68.419,-176.453,7.141,148.302
C03595=1212.659,305.083,-68.390,-176.455,7.138,148.302
C03596=1212.663,304.834,-68.360,-176.457,7.135,148.302
C03597=1212.667,304.586,-68.331,-176.460,7.133,148.302
C03598=1212.672,304.338,-68.300,-176.462,7.130,148.302
C03599=1212.676,304.090,-68.271,-176.464,7.128,148.302
C03600=1212.680,303.842,-68.241,-176.467,7.125,148.302
C03601=1212.685,303.593,-68.212,-176.469,7.123,148.302
C03602=1212.689,303.345,-68.181,-176.472,7.120,148.302
C03603=1212.693,303.097,-68.151,-176.474,7.117,148.302
C03604=1212.698,302.849,-68.122,-176.476,7.115,148.302
C03605=1212.702,302.600,-68.093,-176.479,7.112,148.302
C03606=1212.706,302.352,-68.063,-176.481,7.110,148.302
C03607=1212.711,302.105,-68.033,-176.484,7.107,148.302
C03608=1212.715,301.857,-68.003,-176.486,7.105,148.302
C03609=1212.720,301.608,-67.974,-176.488,7.102,148.302
C03610=1212.724,301.360,-67.944,-176.491,7.099,148.302
C03611=1212.728,301.112,-67.915,-176.493,7.096,148.302
C03612=1212.732,300.864,-67.885,-176.495,7.094,148.303
C03613=1212.737,300.615,-67.855,-176.498,7.091,148.303
C03614=1212.741,300.367,-67.826,-176.501,7.089,148.303
C03615=1212.745,300.119,-67.796,-176.503,7.086,148.303
C03616=1212.750,299.870,-67.767,-176.505,7.084,148.303
C03617=1212.754,299.622,-67.738,-176.508,7.081,148.303
C03618=1212.758,299.374,-67.707,-176.510,7.079,148.303
C03619=1212.762,299.126,-67.678,-176.513,7.076,148.303
C03620=1212.766,298.878,-67.648,-176.515,7.074,148.303
C03621=1212.771,298.630,-67.619,-176.518,7.071,148.303
C03622=1212.775,298.381,-67.591,-176.520,7.068,148.303
C03623=1212.780,298.133,-67.561,-176.522,7.065,148.303
C03624=1212.784,297.884,-67.531,-176.525,7.063,148.303
C03625=1212.789,297.636,-67.502,-176.527,7.060,148.303
C03626=1212.793,297.388,-67.472,-176.530,7.058,148.303
C03627=1212.797,297.140,-67.443,-176.532,7.056,148.304
C03628=1212.801,296.891,-67.413,-176.535,7.053,148.304
C03629=1212.806,296.644,-67.384,-176.537,7.051,148.304
C03630=1212.810,296.396,-67.355,-176.539,7.048,148.304
C03631=1212.814,296.147,-67.325,-176.542,7.046,148.304
C03632=1212.818,295.899,-67.296,-176.544,7.042,148.304
C03633=1212.823,295.650,-67.267,-176.546,7.040,148.304
C03634=1212.827,295.402,-67.238,-176.549,7.037,148.304
C03635=1212.832,295.154,-67.209,-176.552,7.035,148.304
C03636=1212.836,294.906,-67.179,-176.554,7.032,148.304
C03637=1212.839,294.658,-67.150,-176.556,7.030,148.304
C03638=1212.844,294.410,-67.121,-176.559,7.027,148.304
C03639=1212.848,294.161,-67.092,-176.561,7.025,148.304
C03640=1212.852,293.913,-67.063,-176.563,7.023,148.304
C03641=1212.857,293.665,-67.034,-176.567,7.020,148.305
C03642=1212.861,293.417,-67.004,-176.569,7.018,148.305
C03643=1212.866,293.168,-66.975,-176.571,7.015,148.305
C03644=1212.870,292.920,-66.946,-176.573,7.013,148.305
C03645=1212.874,292.671,-66.916,-176.576,7.010,148.305
C03646=1212.879,292.423,-66.888,-176.578,7.007,148.305
C03647=1212.883,292.175,-66.859,-176.581,7.005,148.305
C03648=1212.887,291.927,-66.830,-176.584,7.002,148.305
C03649=1212.891,291.678,-66.801,-176.586,7.000,148.305
C03650=1212.896,291.431,-66.772,-176.588,6.997,148.305
C03651=1212.900,291.182,-66.743,-176.591,6.995,148.305
C03652=1212.905,290.933,-66.714,-176.593,6.992,148.305
